	// OCTAL without notations
	result := stringBuilder.Reset()
		.AddAnyBit(
			anyBit := lwordVar, 
			option := E_AddAnyBitOptions.OCTAL, 
			lowerCase := FALSE, 
			displayedDigitsCount := 64, 
			addNotation := FALSE)
		.Create();
		
	AssertEquals_STRING(
		Actual := result,
		Expected := '0000000000000000000000000000000000000000000000000000000000000253',
		Message := 'Adding lword as OCTAL with addNotation = FALSE was incorrect');
		
	TcUnit.TEST_FINISHED();
END_IF
END_METHOD

METHOD Test28_ANY_REAL_REAL
VAR
	realVar	: REAL := 12345.123888;
	result	: Tc2_System.T_MaxString;
END_VAR
IF TcUnit.TEST_ORDERED('Test28_ANY_REAL_REAL') THEN
	result := stringBuilder.Reset().
		AddAnyReal(
			anyReal := realVar,
			precision := 2,
			round := FALSE)
		.Create();	

	AssertEquals_STRING(
		Actual := result,
		Expected := '12345.12',
		Message := 'Adding REAL with round = FALSE failed.');
		
	result := stringBuilder.Reset().
		AddAnyReal(
			anyReal := realVar,
			precision := 3,
			round := TRUE)
		.Create();	

	AssertEquals_STRING(
		Actual := result,
		Expected := '12345.124',
		Message := 'Adding REAL with round = TRUE failed.');
		
	TcUnit.TEST_FINISHED();
END_IF
END_METHOD

METHOD Test29_ANY_REAL_LREAL
VAR
	lrealVar	: LREAL := 12345.12345678;
	result	: Tc2_System.T_MaxString;
END_VAR
IF TcUnit.TEST_ORDERED('Test29_ANY_REAL_LREAL') THEN
	result := stringBuilder.Reset().
		AddAnyReal(
			anyReal := lrealVar,
			precision := 5,
			round := FALSE)
		.Create();	

	AssertEquals_STRING(
		Actual := result,
		Expected := '12345.12345',
		Message := 'Adding LREAL with round = FALSE failed.');
		
	result := stringBuilder.Reset().
		AddAnyReal(
			anyReal := lrealVar,
			precision := 7,
			round := TRUE)
		.Create();	

	AssertEquals_STRING(
		Actual := result,
		Expected := '12345.1234568',
		Message := 'Adding LREAL with round = TRUE failed.');
		
	TcUnit.TEST_FINISHED();
END_IF
END_METHOD

END_FUNCTION_BLOCK

// ---- TESTS/Test suites/FB_HasTaskInfo_Tests.TcPOU
FUNCTION_BLOCK internal FB_HasTaskInfo_Tests EXTENDS FB_TestSuite
VAR_INPUT
END_VAR
VAR_OUTPUT
END_VAR
VAR
END_VAR

Test01_TaskInfoPropertyValidity();

METHOD Test01_TaskInfoPropertyValidity
VAR_INPUT
END_VAR
VAR_INST
	fbTaskInfo	: FB_HasTaskInfo_ExtensionsForTests;
	cycles	: UINT;
END_VAR
TcUnit.TEST('Test01_TaskInfoPropertyValidity');

AssertTrue(
	Condition := __ISVALIDREF(fbTaskInfo.TaskInfo),
	Message := 'Invalid reference for Taskinfo property. PLC crash will occur if called!');
	
AssertTrue(
	Condition := fbTaskInfo.TaskInfo.AdsPort <> 0,
	Message := 'TaskInfo property is empty.');


TcUnit.TEST_FINISHED();
END_METHOD

END_FUNCTION_BLOCK

// ---- TESTS/Test suites/FB_HasTaskInfo_ExtensionsForTests.TcPOU
// Since FB_HasTaskInfo is an ABSTRACT class, the functionality needs to be implemented by extending the base class
FUNCTION_BLOCK internal FB_HasTaskInfo_ExtensionsForTests EXTENDS FB_HasTaskInfo
VAR_INPUT
END_VAR
VAR_OUTPUT
END_VAR
VAR
END_VAR

END_FUNCTION_BLOCK

// ---- SOURCE/General/FB_HasTaskInfo.TcPOU
{attribute 'no_explicit_call' := 'Body contains no logic, calling methods only allowed.'}
FUNCTION_BLOCK ABSTRACT FB_HasTaskInfo
VAR
	_PlcTaskInfo	: REFERENCE TO PlcTaskSystemInfo;
END_VAR

{attribute 'monitoring':='call'}
PROPERTY TaskInfo : REFERENCE TO PlcTaskSystemInfo
GET
VAR
	taskIndex	: DINT;
END_VAR
IF NOT __ISVALIDREF(_plcTaskInfo) OR_ELSE _plcTaskInfo.CycleTime = 0 THEN
	taskIndex := Tc2_System.GETCURTASKINDEXEX();
	IF taskIndex <> 0 THEN
		_PlcTaskInfo REF= TwinCAT_SystemInfoVarList._TaskInfo[taskIndex];
	END_IF
END_IF

TaskInfo REF= _PlcTaskInfo;
END_GET
END_PROPERTY

END_FUNCTION_BLOCK

// ---- TESTS/Test suites/FB_BoolEx_Tests.TcPOU
FUNCTION_BLOCK INTERNAL FB_BoolEx_Tests EXTENDS FB_TestSuite
VAR_INPUT
END_VAR
VAR_OUTPUT
END_VAR
VAR
	_boolVariable	: BOOL;
	_intVariable	: INT;
	_boolEx			: BoolEx := (variable := _boolVariable);
END_VAR

Test01_BooleanTrue_ExpectTrueAfterElapsedTime();
Test02_BooleanFalse_ExpectTrueAfterElapsedTime();
Test03_RisingAndFallingEdge_ExpectPulses();
Test04_GetAndSetValue();
Test05_Toggle_ExpectValueInverts();
Test06_PulseWithInterval_100ms_ExpectValueChangeEvery100ms();
Test07_Set_ExpectTrue();
Test08_Reset_ExpectFalse();

METHOD Test01_BooleanTrue_ExpectTrueAfterElapsedTime
VAR_INPUT
		
END_VAR
VAR_INST
	boolEx				: BoolEx := (variable := _boolVariable);
	conditionTrueTimer	: Tc2_Standard.TON;
END_VAR
TcUnit.TEST('Test01_BooleanTrue_ExpectTrueAfterElapsedTime');

conditionTrueTimer();
IF NOT conditionTrueTimer.Q THEN
	_boolVariable := TRUE;
	conditionTrueTimer(IN := TRUE, PT := T#20MS);
	AssertFalse(
		Condition := boolEx.HasBeenTrueForAtLeast(T#20MS),
		Message := 'HasBeenTrueForAtLeast returned TRUE before elapsed time.');
ELSE
	AssertTrue(
		Condition := boolEx.HasBeenTrueForAtLeast(T#20MS),
		Message := 'HasBeenTrueForAtLeast returned FALSE after elapsed time.');
		TcUnit.TEST_FINISHED();
END_IF
END_METHOD

METHOD Test02_BooleanFalse_ExpectTrueAfterElapsedTime : BOOL
VAR_INST
	boolEx			: BoolEx := (variable := _boolVariable);
	conditionTimer	: Tc2_Standard.TON;
END_VAR
TcUnit.TEST('Test02_BooleanFalse_ExpectTrueAfterElapsedTime');
IF TcUnit.IS_TEST_FINISHED('Test01_BooleanTrue_ExpectTrueAfterElapsedTime') THEN
	_boolVariable := FALSE;
	conditionTimer();
	IF NOT conditionTimer.Q THEN
		conditionTimer(IN := TRUE, PT := T#20MS);
		AssertFalse(
			Condition := boolEx.HasBeenFalseForAtLeast(T#20MS),
			Message := 'HasBeenFalseForAtLeast returned TRUE before elapsed time.');
	ELSE
		AssertTrue(
			Condition := boolEx.HasBeenFalseForAtLeast(T#20MS),
			Message := 'HasBeenFalseForAtLeast returned FALSE after elapsed time.');
			TcUnit.TEST_FINISHED();
	END_IF
END_IF
END_METHOD

METHOD Test03_RisingAndFallingEdge_ExpectPulses
VAR_INPUT
END_VAR

VAR_INST
	boolEx : BoolEx := (variable := _boolVariable);
END_VAR
TcUnit.TEST('Test03_RisingAndFallingEdge_ExpectPulses');


IF TcUnit.IS_TEST_FINISHED('Test02_BooleanFalse_ExpectTrueAfterElapsedTime') THEN
	_boolVariable := FALSE;
	AssertFalse(
		Condition := boolEx.HasRisingEdge,
		Message := 'When value has not changed, the HasRisingEdge should be false');
	AssertFalse(
		Condition := boolEx.HasFallingEdge,
		Message := 'When value has not changed, the HasFallingEdge should be false');
	_boolVariable := TRUE;	
	AssertTrue(
		Condition := boolEx.HasRisingEdge,
		Message := 'When value has changed from FALSE to TRUE, the HasRisingEdge should be TRUE');
	AssertFalse(
		Condition := boolEx.HasFallingEdge,
		Message := 'When value has changed to TRUE, the HasFallingEdge should be false');
	_boolVariable := FALSE;
	AssertTrue(
		Condition := boolEx.HasFallingEdge,
		Message := 'When value has changed from TRUE to FALSE, the HasFallingEdge should be TRUE');
	AssertFalse(
		Condition := boolEx.HasRisingEdge,
		Message := 'When value has not changed, the HasRisingEdge should be false');
	AssertFalse(
		Condition := boolEx.HasFallingEdge,
		Message := 'When value has not changed, the HasRisingEdge should be false');	
	TcUnit.TEST_FINISHED();
	
END_IF
END_METHOD

METHOD Test04_GetAndSetValue
VAR_INPUT
END_VAR
VAR_INST
	boolEx	: BoolEx := (variable := _boolVariable);
END_VAR
TcUnit.TEST('Test04_GetAndSetValue');
IF TcUnit.IS_TEST_FINISHED('Test03_RisingAndFallingEdge_ExpectPulses') THEN
	_boolVariable := FALSE;
	boolEx.Value := TRUE;	
	AssertTrue(
		Condition := _boolVariable,
		Message := 'Setting value to TRUE failed');
		
	boolEx.Value := FALSE;
	AssertFalse(
		Condition := _boolVariable,
		Message := 'Setting value to FALSE failed');
		
	AssertEquals_BOOL(
		Actual := boolEx.Value,
		Expected := _boolVariable,
		Message := 'Value returned incorrect result.');
		
	_boolVariable := TRUE;
	AssertEquals_BOOL(
		Actual := boolEx.Value,
		Expected := _boolVariable,
		Message := 'Value returned incorrect result.');
	
	TcUnit.TEST_FINISHED();
END_IF
END_METHOD

METHOD Test05_Toggle_ExpectValueInverts
VAR_INPUT
END_VAR
TcUnit.TEST('Test05_Toggle_ExpectValueInverts');
IF TcUnit.IS_TEST_FINISHED('Test04_GetAndSetValue') THEN
	_boolEx.Value := FALSE;
	AssertFalse(
		Condition := _boolEx.Value,
		Message := 'Expected value to be false.');
		
	_boolEx.Toggle();
	AssertTrue(
		Condition := _boolEx.Value,
		Message := 'Toggle to TRUE failed');
		
	_boolEx.Toggle();
	AssertFalse(
		Condition := _boolEx.Value,
		Message := 'Toggle to FALSE failed');	
	TcUnit.TEST_FINISHED();
END_IF
END_METHOD

METHOD Test06_PulseWithInterval_100ms_ExpectValueChangeEvery100ms
VAR_INPUT
END_VAR
VAR_INST
	timerOn		: Tc2_Standard.TON;
	timerOff	: Tc2_Standard.TON;
END_VAR
TcUnit.TEST('Test06_PulseWithInterval_100ms_ExpectValueChangeEvery100ms');
IF TcUnit.IS_TEST_FINISHED('Test05_Toggle_ExpectValueInverts') THEN
	_boolEx.Value := FALSE;
	_boolEx.PulseWithInterval(durationOn := T#100MS, durationOff := T#50MS);
	timerOn(IN := TRUE, PT := T#100MS);
	IF NOT timerOn.Q THEN
		AssertTrue(
			Condition := _boolEx.Value,
			Message := 'Value should be TRUE until the durationOn expires.');
	ELSE
		timerOff(IN := TRUE, PT := T#50MS);
		IF timeroff.Q THEN
			AssertTrue(
				Condition := _boolEx.Value,
				Message := 'Value should be TRUE after the durationOff expires.');
			TcUnit.TEST_FINISHED();
			RETURN;
		END_IF
		AssertFalse(
			Condition := _boolEx.Value,
			Message := 'Value should be FALSE after durationOn expires.');

	END_IF
END_IF
END_METHOD

METHOD Test07_Set_ExpectTrue
VAR_INPUT
END_VAR
TcUnit.TEST('Test07_Set_ExpectTrue');

IF TcUnit.IS_TEST_FINISHED('Test06_PulseWithInterval_100ms_ExpectValueChangeEvery100ms') THEN 
	_boolEx.Value := FALSE;
	_boolEx.Set();
	AssertTrue(
		Condition := _boolEx.Value,
		Message := 'Set() did not set the value to TRUE.');
	TcUnit.TEST_FINISHED();
END_IF
END_METHOD

METHOD Test08_Reset_ExpectFalse
VAR_INPUT
END_VAR
TcUnit.TEST('Test08_Reset_ExpectFalse');

IF TcUnit.IS_TEST_FINISHED('Test07_Set_ExpectTrue') THEN 
	_boolEx.Value := TRUE;
	_boolEx.Reset();
	AssertFalse(
		Condition := _boolEx.Value,
		Message := 'Reset() did not set the value to FALSE.');
	TcUnit.TEST_FINISHED();
END_IF
END_METHOD

END_FUNCTION_BLOCK

// ---- SOURCE/General/Variable extensions/BoolEx.TcPOU
// An extension to boolean variable
FUNCTION_BLOCK BoolEx
VAR_INPUT
	variable			: REFERENCE TO BOOL;
END_VAR

VAR
	
	_risingEdge			: Tc2_Standard.R_TRIG;
	_fallingEdge		: Tc2_Standard.F_TRIG;
	afterinitvarinfo 	: ST_VarInfo;
END_VAR

// Returns TRUE if monitored value has been FALSE for at lease for the provided "duration"
METHOD HasBeenFalseForAtLeast : BOOL
VAR_INPUT
	duration	: TIME;
END_VAR

VAR_INST
	timer	: Tc2_Standard.TON;

END_VAR
IF NOT IsVarValid() THEN
	RETURN;
END_IF

timer(IN := NOT variable, PT := duration);
HasBeenFalseForAtLeast := timer.Q;
END_METHOD

// Returns TRUE if monitored value has been TRUE for at lease for the provided "duration"
METHOD HasBeenTrueForAtLeast : BOOL
VAR_INPUT
	duration	: TIME;
END_VAR

VAR_INST
	timer	: Tc2_Standard.TON;
	ptrBool	: POINTER TO BOOL;
END_VAR
IF NOT IsVarValid() THEN
	RETURN;
END_IF

timer(IN := variable, PT := duration);
HasBeenTrueForAtLeast := timer.Q;
END_METHOD

// Returns TRUE if oberved variable change from TRUE to FALSE from the last call.
PROPERTY HasFallingEdge : BOOL
GET
_fallingEdge(CLK := variable);
HasFallingEdge := _fallingEdge.Q;
END_GET
END_PROPERTY

// Returns TRUE if oberved variable change from FALSE to TRUE from the last call.
PROPERTY HasRisingEdge : BOOL
GET
_risingEdge(CLK := variable);
HasRisingEdge := _risingEdge.Q;
END_GET
END_PROPERTY

METHOD PROTECTED IsVarValid : BOOL
IsVarValid := __ISVALIDREF(variable);
END_METHOD

// Pulses the virabile (TRUE/FALSE) with the provided on and off duration
METHOD PulseWithInterval
VAR_INPUT
	durationOn	: TIME;
	durationOff	: TIME;
END_VAR
VAR_INST
	timerOn		: Tc2_Standard.TON;
	timerOff	: Tc2_Standard.TON;
END_VAR
IF NOT IsVarValid() THEN
	RETURN;
END_IF
// In order to properly trigger immediate change, call both timers twice. 
// This way when ON is elapsed, OFF starts imediately and vice versa.
timerOff(IN := timerOn.Q, PT := durationOff);
timerOn(IN := NOT timerOff.Q, PT := durationOn);
timerOff(IN := timerOn.Q, PT := durationOff);
timerOn(IN := NOT timerOff.Q, PT := durationOn);
variable := NOT timerOn.Q;
END_METHOD

// Sets the value to FALSE
METHOD Reset
VAR_INPUT
END_VAR
IF NOT IsVarValid() THEN
	RETURN;
END_IF

variable := FALSE;
END_METHOD

// Sets the value to TRUE
METHOD Set
VAR_INPUT
END_VAR
IF NOT IsVarValid() THEN
	RETURN;
END_IF

variable := TRUE;
END_METHOD

METHOD Toggle
IF NOT IsVarValid() THEN
	RETURN;
END_IF

variable := NOT variable;
END_METHOD

PROPERTY Value : BOOL
GET
Value := variable;
END_GET
SET
variable := Value;
END_SET
END_PROPERTY

END_FUNCTION_BLOCK

// ---- TESTS/Test suites/FB_EthercatHelper_Tests.TcPOU
FUNCTION_BLOCK INTERNAL FB_EthercatHelper_Tests EXTENDS FB_TestSuite
VAR_INPUT
END_VAR
VAR_OUTPUT
END_VAR
VAR
END_VAR

Test01_ConvertBeckhoffEcState_ProvideAllOptions_ExpectCorrectResults();

METHOD Test01_ConvertBeckhoffEcState_ProvideAllOptions_ExpectCorrectResults
VAR_INST
	ecSlaveState		: Tc2_EtherCAT.ST_EcSlaveState;
	helperEcSlaveState	: ST_EcSlaveState;
END_VAR
TcUnit.TEST('Test01_ConvertBeckhoffEcState_ProvideAllOptions_ExpectCorrectResults');

// Init
ecSlaveState.deviceState := Tc2_EtherCAT.EC_DEVICE_STATE_INIT;
helperEcSlaveState := EthercatHelper.ConvertBeckhoffEcStateToCustomStruct(ecSlaveState);
AssertEquals_BYTE(Tc2_EtherCAT.EC_DEVICE_STATE_INIT, helperEcSlaveState.Device.State, 'Incorrect state for EC_DEVICE_STATE_INIT.');
AssertEquals_BYTE(E_EcDeviceStateExtras.NOTHING, helperEcSlaveState.Device.StateExtras, 'EC_DEVICE_STATE_INIT - Extras NOTHING expected');
	
ecSlaveState.deviceState := Tc2_EtherCAT.EC_DEVICE_STATE_INIT OR Tc2_EtherCAT.EC_DEVICE_STATE_INITCMD_ERROR;
helperEcSlaveState := EthercatHelper.ConvertBeckhoffEcStateToCustomStruct(ecSlaveState);
AssertEquals_BYTE(Tc2_EtherCAT.EC_DEVICE_STATE_INIT, helperEcSlaveState.Device.State,'Incorrect state for EC_DEVICE_STATE_INIT OR EC_DEVICE_STATE_INITCMD_ERROR');
AssertEquals_BYTE(E_EcDeviceStateExtras.INIIT_CMD_ERROR, helperEcSlaveState.Device.StateExtras, 'EC_DEVICE_STATE_INIT - Extras INIIT_CMD_ERROR expected');
	
ecSlaveState.deviceState := Tc2_EtherCAT.EC_DEVICE_STATE_INIT OR Tc2_EtherCAT.EC_DEVICE_STATE_INVALID_VPRS;
helperEcSlaveState := EthercatHelper.ConvertBeckhoffEcStateToCustomStruct(ecSlaveState);
AssertEquals_BYTE(Tc2_EtherCAT.EC_DEVICE_STATE_INIT, helperEcSlaveState.Device.State,'Incorrect state for EC_DEVICE_STATE_INIT OR EC_DEVICE_STATE_INVALID_VPRS');
AssertEquals_BYTE(E_EcDeviceStateExtras.INVALID_VPRS, helperEcSlaveState.Device.StateExtras, 'EC_DEVICE_STATE_INIT - Extras INVALID_VPRS expected');

ecSlaveState.deviceState := Tc2_EtherCAT.EC_DEVICE_STATE_INIT OR Tc2_EtherCAT.EC_DEVICE_STATE_DISABLED;
helperEcSlaveState := EthercatHelper.ConvertBeckhoffEcStateToCustomStruct(ecSlaveState);
AssertEquals_BYTE(Tc2_EtherCAT.EC_DEVICE_STATE_INIT, helperEcSlaveState.Device.State,'Incorrect state for EC_DEVICE_STATE_INIT OR EC_DEVICE_STATE_DISABLED');
AssertEquals_BYTE(E_EcDeviceStateExtras.DISABLED, helperEcSlaveState.Device.StateExtras, 'EC_DEVICE_STATE_INIT - Extras DISABLED expected');

ecSlaveState.deviceState := Tc2_EtherCAT.EC_DEVICE_STATE_INIT OR Tc2_EtherCAT.EC_DEVICE_STATE_ERROR;
helperEcSlaveState := EthercatHelper.ConvertBeckhoffEcStateToCustomStruct(ecSlaveState);
AssertEquals_BYTE(Tc2_EtherCAT.EC_DEVICE_STATE_INIT, helperEcSlaveState.Device.State,'Incorrect state for EC_DEVICE_STATE_INIT OR EC_DEVICE_STATE_ERROR');
AssertEquals_BYTE(E_EcDeviceStateExtras.STATE_MACHINE_ERROR, helperEcSlaveState.Device.StateExtras, 'EC_DEVICE_STATE_INIT - Extras STATE_MACHINE_ERROR expected');
	
// Pre-op
ecSlaveState.deviceState := Tc2_EtherCAT.EC_DEVICE_STATE_PREOP;
helperEcSlaveState := EthercatHelper.ConvertBeckhoffEcStateToCustomStruct(ecSlaveState);
AssertEquals_BYTE(Tc2_EtherCAT.EC_DEVICE_STATE_PREOP, helperEcSlaveState.Device.State, 'Incorrect state for EC_DEVICE_STATE_PREOP.');
AssertEquals_BYTE(E_EcDeviceStateExtras.NOTHING, helperEcSlaveState.Device.StateExtras, 'EC_DEVICE_STATE_PREOP - Extras NOTHING expected');
	
ecSlaveState.deviceState := Tc2_EtherCAT.EC_DEVICE_STATE_PREOP OR Tc2_EtherCAT.EC_DEVICE_STATE_INITCMD_ERROR;
helperEcSlaveState := EthercatHelper.ConvertBeckhoffEcStateToCustomStruct(ecSlaveState);
AssertEquals_BYTE(Tc2_EtherCAT.EC_DEVICE_STATE_PREOP, helperEcSlaveState.Device.State,'Incorrect state for EC_DEVICE_STATE_PREOP OR EC_DEVICE_STATE_INITCMD_ERROR');
AssertEquals_BYTE(E_EcDeviceStateExtras.INIIT_CMD_ERROR, helperEcSlaveState.Device.StateExtras, 'EC_DEVICE_STATE_PREOP - Extras INIIT_CMD_ERROR expected');
	
ecSlaveState.deviceState := Tc2_EtherCAT.EC_DEVICE_STATE_PREOP OR Tc2_EtherCAT.EC_DEVICE_STATE_INVALID_VPRS;
helperEcSlaveState := EthercatHelper.ConvertBeckhoffEcStateToCustomStruct(ecSlaveState);
AssertEquals_BYTE(Tc2_EtherCAT.EC_DEVICE_STATE_PREOP, helperEcSlaveState.Device.State,'Incorrect state for EC_DEVICE_STATE_PREOP OR EC_DEVICE_STATE_INVALID_VPRS');
AssertEquals_BYTE(E_EcDeviceStateExtras.INVALID_VPRS, helperEcSlaveState.Device.StateExtras, 'EC_DEVICE_STATE_PREOP - Extras INVALID_VPRS expected');

ecSlaveState.deviceState := Tc2_EtherCAT.EC_DEVICE_STATE_PREOP OR Tc2_EtherCAT.EC_DEVICE_STATE_DISABLED;
helperEcSlaveState := EthercatHelper.ConvertBeckhoffEcStateToCustomStruct(ecSlaveState);
AssertEquals_BYTE(Tc2_EtherCAT.EC_DEVICE_STATE_PREOP, helperEcSlaveState.Device.State,'Incorrect state for EC_DEVICE_STATE_PREOP OR EC_DEVICE_STATE_DISABLED');
AssertEquals_BYTE(E_EcDeviceStateExtras.DISABLED, helperEcSlaveState.Device.StateExtras, 'EC_DEVICE_STATE_PREOP - Extras DISABLED expected');

ecSlaveState.deviceState := Tc2_EtherCAT.EC_DEVICE_STATE_PREOP OR Tc2_EtherCAT.EC_DEVICE_STATE_ERROR;
helperEcSlaveState := EthercatHelper.ConvertBeckhoffEcStateToCustomStruct(ecSlaveState);
AssertEquals_BYTE(Tc2_EtherCAT.EC_DEVICE_STATE_PREOP, helperEcSlaveState.Device.State,'Incorrect state for EC_DEVICE_STATE_PREOP OR EC_DEVICE_STATE_ERROR');
AssertEquals_BYTE(E_EcDeviceStateExtras.STATE_MACHINE_ERROR, helperEcSlaveState.Device.StateExtras, 'EC_DEVICE_STATE_PREOP - Extras STATE_MACHINE_ERROR expected');

// Bootstrap
ecSlaveState.deviceState := Tc2_EtherCAT.EC_DEVICE_STATE_BOOTSTRAP;
helperEcSlaveState := EthercatHelper.ConvertBeckhoffEcStateToCustomStruct(ecSlaveState);
AssertEquals_BYTE(Tc2_EtherCAT.EC_DEVICE_STATE_BOOTSTRAP, helperEcSlaveState.Device.State, 'Incorrect state for EC_DEVICE_STATE_BOOTSTRAP.');
AssertEquals_BYTE(E_EcDeviceStateExtras.NOTHING, helperEcSlaveState.Device.StateExtras, 'EC_DEVICE_STATE_BOOTSTRAP - Extras NOTHING expected');
	
ecSlaveState.deviceState := Tc2_EtherCAT.EC_DEVICE_STATE_BOOTSTRAP OR Tc2_EtherCAT.EC_DEVICE_STATE_INITCMD_ERROR;
helperEcSlaveState := EthercatHelper.ConvertBeckhoffEcStateToCustomStruct(ecSlaveState);
AssertEquals_BYTE(Tc2_EtherCAT.EC_DEVICE_STATE_BOOTSTRAP, helperEcSlaveState.Device.State,'Incorrect state for EC_DEVICE_STATE_BOOTSTRAP OR EC_DEVICE_STATE_INITCMD_ERROR');
AssertEquals_BYTE(E_EcDeviceStateExtras.INIIT_CMD_ERROR, helperEcSlaveState.Device.StateExtras, 'EC_DEVICE_STATE_BOOTSTRAP - Extras INIIT_CMD_ERROR expected');
	
ecSlaveState.deviceState := Tc2_EtherCAT.EC_DEVICE_STATE_BOOTSTRAP OR Tc2_EtherCAT.EC_DEVICE_STATE_INVALID_VPRS;
helperEcSlaveState := EthercatHelper.ConvertBeckhoffEcStateToCustomStruct(ecSlaveState);
AssertEquals_BYTE(Tc2_EtherCAT.EC_DEVICE_STATE_BOOTSTRAP, helperEcSlaveState.Device.State,'Incorrect state for EC_DEVICE_STATE_BOOTSTRAP OR EC_DEVICE_STATE_INVALID_VPRS');
AssertEquals_BYTE(E_EcDeviceStateExtras.INVALID_VPRS, helperEcSlaveState.Device.StateExtras, 'EC_DEVICE_STATE_BOOTSTRAP - Extras INVALID_VPRS expected');

ecSlaveState.deviceState := Tc2_EtherCAT.EC_DEVICE_STATE_BOOTSTRAP OR Tc2_EtherCAT.EC_DEVICE_STATE_DISABLED;
helperEcSlaveState := EthercatHelper.ConvertBeckhoffEcStateToCustomStruct(ecSlaveState);
AssertEquals_BYTE(Tc2_EtherCAT.EC_DEVICE_STATE_BOOTSTRAP, helperEcSlaveState.Device.State,'Incorrect state for EC_DEVICE_STATE_BOOTSTRAP OR EC_DEVICE_STATE_DISABLED');
AssertEquals_BYTE(E_EcDeviceStateExtras.DISABLED, helperEcSlaveState.Device.StateExtras, 'EC_DEVICE_STATE_BOOTSTRAP - Extras DISABLED expected');

ecSlaveState.deviceState := Tc2_EtherCAT.EC_DEVICE_STATE_BOOTSTRAP OR Tc2_EtherCAT.EC_DEVICE_STATE_ERROR;
helperEcSlaveState := EthercatHelper.ConvertBeckhoffEcStateToCustomStruct(ecSlaveState);
AssertEquals_BYTE(Tc2_EtherCAT.EC_DEVICE_STATE_BOOTSTRAP, helperEcSlaveState.Device.State,'Incorrect state for EC_DEVICE_STATE_BOOTSTRAP OR EC_DEVICE_STATE_ERROR');
AssertEquals_BYTE(E_EcDeviceStateExtras.STATE_MACHINE_ERROR, helperEcSlaveState.Device.StateExtras, 'EC_DEVICE_STATE_BOOTSTRAP - Extras STATE_MACHINE_ERROR expected');

// Safeop
ecSlaveState.deviceState := Tc2_EtherCAT.EC_DEVICE_STATE_SAFEOP;
helperEcSlaveState := EthercatHelper.ConvertBeckhoffEcStateToCustomStruct(ecSlaveState);
AssertEquals_BYTE(Tc2_EtherCAT.EC_DEVICE_STATE_SAFEOP, helperEcSlaveState.Device.State, 'Incorrect state for EC_DEVICE_STATE_SAFEOP.');
AssertEquals_BYTE(E_EcDeviceStateExtras.NOTHING, helperEcSlaveState.Device.StateExtras, 'EC_DEVICE_STATE_SAFEOP - Extras NOTHING expected');
	
ecSlaveState.deviceState := Tc2_EtherCAT.EC_DEVICE_STATE_SAFEOP OR Tc2_EtherCAT.EC_DEVICE_STATE_INITCMD_ERROR;
helperEcSlaveState := EthercatHelper.ConvertBeckhoffEcStateToCustomStruct(ecSlaveState);
AssertEquals_BYTE(Tc2_EtherCAT.EC_DEVICE_STATE_SAFEOP, helperEcSlaveState.Device.State,'Incorrect state for EC_DEVICE_STATE_BOOTSTRAP OR EC_DEVICE_STATE_INITCMD_ERROR');
AssertEquals_BYTE(E_EcDeviceStateExtras.INIIT_CMD_ERROR, helperEcSlaveState.Device.StateExtras, 'EC_DEVICE_STATE_SAFEOP - Extras INIIT_CMD_ERROR expected');
	
ecSlaveState.deviceState := Tc2_EtherCAT.EC_DEVICE_STATE_SAFEOP OR Tc2_EtherCAT.EC_DEVICE_STATE_INVALID_VPRS;
helperEcSlaveState := EthercatHelper.ConvertBeckhoffEcStateToCustomStruct(ecSlaveState);
AssertEquals_BYTE(Tc2_EtherCAT.EC_DEVICE_STATE_SAFEOP, helperEcSlaveState.Device.State,'Incorrect state for EC_DEVICE_STATE_SAFEOP OR EC_DEVICE_STATE_INVALID_VPRS');
AssertEquals_BYTE(E_EcDeviceStateExtras.INVALID_VPRS, helperEcSlaveState.Device.StateExtras, 'EC_DEVICE_STATE_SAFEOP - Extras INVALID_VPRS expected');

ecSlaveState.deviceState := Tc2_EtherCAT.EC_DEVICE_STATE_SAFEOP OR Tc2_EtherCAT.EC_DEVICE_STATE_DISABLED;
helperEcSlaveState := EthercatHelper.ConvertBeckhoffEcStateToCustomStruct(ecSlaveState);
AssertEquals_BYTE(Tc2_EtherCAT.EC_DEVICE_STATE_SAFEOP, helperEcSlaveState.Device.State,'Incorrect state for EC_DEVICE_STATE_SAFEOP OR EC_DEVICE_STATE_DISABLED');
AssertEquals_BYTE(E_EcDeviceStateExtras.DISABLED, helperEcSlaveState.Device.StateExtras, 'EC_DEVICE_STATE_SAFEOP - Extras DISABLED expected');

ecSlaveState.deviceState := Tc2_EtherCAT.EC_DEVICE_STATE_SAFEOP OR Tc2_EtherCAT.EC_DEVICE_STATE_ERROR;
helperEcSlaveState := EthercatHelper.ConvertBeckhoffEcStateToCustomStruct(ecSlaveState);
AssertEquals_BYTE(Tc2_EtherCAT.EC_DEVICE_STATE_SAFEOP, helperEcSlaveState.Device.State,'Incorrect state for EC_DEVICE_STATE_SAFEOP OR EC_DEVICE_STATE_ERROR');
AssertEquals_BYTE(E_EcDeviceStateExtras.STATE_MACHINE_ERROR, helperEcSlaveState.Device.StateExtras, 'EC_DEVICE_STATE_SAFEOP - Extras STATE_MACHINE_ERROR expected');

// OP
ecSlaveState.deviceState := Tc2_EtherCAT.EC_DEVICE_STATE_OP;
helperEcSlaveState := EthercatHelper.ConvertBeckhoffEcStateToCustomStruct(ecSlaveState);
AssertEquals_BYTE(Tc2_EtherCAT.EC_DEVICE_STATE_OP, helperEcSlaveState.Device.State, 'Incorrect state for EC_DEVICE_STATE_OP.');
AssertEquals_BYTE(E_EcDeviceStateExtras.NOTHING, helperEcSlaveState.Device.StateExtras, 'EC_DEVICE_STATE_OP - Extras NOTHING expected');
	
ecSlaveState.deviceState := Tc2_EtherCAT.EC_DEVICE_STATE_OP OR Tc2_EtherCAT.EC_DEVICE_STATE_INITCMD_ERROR;
helperEcSlaveState := EthercatHelper.ConvertBeckhoffEcStateToCustomStruct(ecSlaveState);
AssertEquals_BYTE(Tc2_EtherCAT.EC_DEVICE_STATE_OP, helperEcSlaveState.Device.State,'Incorrect state for EC_DEVICE_STATE_OP OR EC_DEVICE_STATE_INITCMD_ERROR');
AssertEquals_BYTE(E_EcDeviceStateExtras.INIIT_CMD_ERROR, helperEcSlaveState.Device.StateExtras, 'EC_DEVICE_STATE_OP - Extras INIIT_CMD_ERROR expected');
	
ecSlaveState.deviceState := Tc2_EtherCAT.EC_DEVICE_STATE_OP OR Tc2_EtherCAT.EC_DEVICE_STATE_INVALID_VPRS;
helperEcSlaveState := EthercatHelper.ConvertBeckhoffEcStateToCustomStruct(ecSlaveState);
AssertEquals_BYTE(Tc2_EtherCAT.EC_DEVICE_STATE_OP, helperEcSlaveState.Device.State,'Incorrect state for EC_DEVICE_STATE_OP OR EC_DEVICE_STATE_INVALID_VPRS');
AssertEquals_BYTE(E_EcDeviceStateExtras.INVALID_VPRS, helperEcSlaveState.Device.StateExtras, 'EC_DEVICE_STATE_OP - Extras INVALID_VPRS expected');

ecSlaveState.deviceState := Tc2_EtherCAT.EC_DEVICE_STATE_OP OR Tc2_EtherCAT.EC_DEVICE_STATE_DISABLED;
helperEcSlaveState := EthercatHelper.ConvertBeckhoffEcStateToCustomStruct(ecSlaveState);
AssertEquals_BYTE(Tc2_EtherCAT.EC_DEVICE_STATE_OP, helperEcSlaveState.Device.State,'Incorrect state for EC_DEVICE_STATE_OP OR EC_DEVICE_STATE_DISABLED');
AssertEquals_BYTE(E_EcDeviceStateExtras.DISABLED, helperEcSlaveState.Device.StateExtras, 'EC_DEVICE_STATE_OP - Extras DISABLED expected');

ecSlaveState.deviceState := Tc2_EtherCAT.EC_DEVICE_STATE_OP OR Tc2_EtherCAT.EC_DEVICE_STATE_ERROR;
helperEcSlaveState := EthercatHelper.ConvertBeckhoffEcStateToCustomStruct(ecSlaveState);
AssertEquals_BYTE(Tc2_EtherCAT.EC_DEVICE_STATE_OP, helperEcSlaveState.Device.State,'Incorrect state for EC_DEVICE_STATE_OP OR EC_DEVICE_STATE_ERROR');
AssertEquals_BYTE(E_EcDeviceStateExtras.STATE_MACHINE_ERROR, helperEcSlaveState.Device.StateExtras, 'EC_DEVICE_STATE_OP - Extras STATE_MACHINE_ERROR expected');

// Link state

//EC_LINK_STATE_OK
ecSlaveState.linkState := Tc2_EtherCAT.EC_LINK_STATE_OK;
helperEcSlaveState := EthercatHelper.ConvertBeckhoffEcStateToCustomStruct(ecSlaveState);
AssertEquals_BYTE(Tc2_EtherCAT.EC_LINK_STATE_OK, helperEcSlaveState.Link, 'Invalid link state for EC_LINK_STATE_OK');

// EC_LINK_STATE_ADDITIONAL_LINK
ecSlaveState.linkState := Tc2_EtherCAT.EC_LINK_STATE_ADDITIONAL_LINK;
helperEcSlaveState := EthercatHelper.ConvertBeckhoffEcStateToCustomStruct(ecSlaveState);
AssertEquals_BYTE(E_EcLinkState.ADDITIONAL_LINK, helperEcSlaveState.Link, 'Invalid link state for EC_LINK_STATE_ADDITIONAL_LINK');

// EC_LINK_STATE_LINK_WITHOUT_COMM
ecSlaveState.linkState := Tc2_EtherCAT.EC_LINK_STATE_LINK_WITHOUT_COMM;
helperEcSlaveState := EthercatHelper.ConvertBeckhoffEcStateToCustomStruct(ecSlaveState);
AssertEquals_BYTE(E_EcLinkState.LINK_WITHOUT_COMM, helperEcSlaveState.Link, 'Invalid link state for EC_LINK_STATE_LINK_WITHOUT_COMM');

// EC_LINK_STATE_MISSING_LINK
ecSlaveState.linkState := Tc2_EtherCAT.EC_LINK_STATE_MISSING_LINK;
helperEcSlaveState := EthercatHelper.ConvertBeckhoffEcStateToCustomStruct(ecSlaveState);
AssertEquals_BYTE(E_EcLinkState.MISSING_LINK, helperEcSlaveState.Link, 'Invalid link state for EC_LINK_STATE_MISSING_LINK');

// EC_LINK_STATE_NOT_PRESENT
ecSlaveState.linkState := Tc2_EtherCAT.EC_LINK_STATE_NOT_PRESENT;
helperEcSlaveState := EthercatHelper.ConvertBeckhoffEcStateToCustomStruct(ecSlaveState);
AssertEquals_BYTE(E_EcLinkState.NOT_PRESENT, helperEcSlaveState.Link, 'Invalid link state for EC_LINK_STATE_NOT_PRESENT');

// EC_LINK_STATE_PORT_A
ecSlaveState.linkState := Tc2_EtherCAT.EC_LINK_STATE_PORT_A;
helperEcSlaveState := EthercatHelper.ConvertBeckhoffEcStateToCustomStruct(ecSlaveState);
AssertEquals_BYTE(E_EcLinkState.PORT_A, helperEcSlaveState.Link, 'Invalid link state for EC_LINK_STATE_PORT_A');

// EC_LINK_STATE_PORT_B
ecSlaveState.linkState := Tc2_EtherCAT.EC_LINK_STATE_PORT_B;
helperEcSlaveState := EthercatHelper.ConvertBeckhoffEcStateToCustomStruct(ecSlaveState);
AssertEquals_BYTE(E_EcLinkState.PORT_B, helperEcSlaveState.Link, 'Invalid link state for EC_LINK_STATE_PORT_B');

// EC_LINK_STATE_PORT_C
ecSlaveState.linkState := Tc2_EtherCAT.EC_LINK_STATE_PORT_C;
helperEcSlaveState := EthercatHelper.ConvertBeckhoffEcStateToCustomStruct(ecSlaveState);
AssertEquals_BYTE(E_EcLinkState.PORT_C, helperEcSlaveState.Link, 'Invalid link state for EC_LINK_STATE_PORT_C');

// EC_LINK_STATE_PORT_D
ecSlaveState.linkState := Tc2_EtherCAT.EC_LINK_STATE_PORT_D;
helperEcSlaveState := EthercatHelper.ConvertBeckhoffEcStateToCustomStruct(ecSlaveState);
AssertEquals_BYTE(E_EcLinkState.PORT_D, helperEcSlaveState.Link, 'Invalid link state for EC_LINK_STATE_PORT_D');

TcUnit.TEST_FINISHED();
END_METHOD

END_FUNCTION_BLOCK

// ---- SOURCE/Beckhoff/EtherCAT/EthercatHelper.TcPOU
{attribute 'hide_all_locals'}
PROGRAM EthercatHelper
VAR
	fbReadDeviceName	: Tc2_IoFunctions.IOF_GetBoxNameByAddr;
	nMasterId			: UDINT;
END_VAR

// Converts Tc2_EtherCAT.ST_EcSlaveState to ZigaLibs_Core.ST_EcSlaveState and returns the converted structure.
METHOD ConvertBeckhoffEcStateToCustomStruct : ST_EcSlaveState
VAR_INPUT
	ecSlaveState	: Tc2_EtherCAT.ST_EcSlaveState;
END_VAR
VAR CONSTANT
	SLAVE_STATE_MASK 		: BYTE := 16#0F;
	SLAVE_STATE_EXTRAS_MASK : BYTE := 16#F0;
END_VAR
ConvertBeckhoffEcStateToCustomStruct.Device.State := SLAVE_STATE_MASK AND ecSlaveState.deviceState;
ConvertBeckhoffEcStateToCustomStruct.Device.StateExtras := SLAVE_STATE_EXTRAS_MASK AND ecSlaveState.deviceState;
ConvertBeckhoffEcStateToCustomStruct.Link := ecSlaveState.linkState;
END_METHOD

METHOD PUBLIC GetBoxNameByAddress : T_MaxString
VAR_INPUT
	PlcRuntimeNetId		: Tc2_System.T_AmsNetID; // NetId of the PLC where the devuce is located
	AmsNetId			: AMSADDR; // NetId of the box
	outError			: REFERENCE TO BOOL;	// If an error occurs while executing, method will provide the error flag here. This is a pointer to YOUR boolean error variable.
END_VAR

VAR
	sNetId	: Tc2_System.T_AmsNetID;
END_VAR
sNetId := AdsHelper.NetIdToString(AmsNetId.netId);
fbReadDeviceName(
	NETID := PlcRuntimeNetId,
	DEVICEID := AdsHelper.GetEthercatMasterIdFromNetIdString(netId := sNetId),
	BOXADDR := AmsNetId.port,
	START := NOT fbReadDeviceName.BUSY);
	
outError := fbReadDeviceName.ERR;
GetBoxNameByAddress := fbReadDeviceName.BOXNAME;
END_METHOD

END_PROGRAM

// ---- TESTS/Test suites/FB_Malloc_Tests.TcPOU
FUNCTION_BLOCK internal FB_Malloc_Tests EXTENDS FB_TestSuite
VAR_INPUT
END_VAR
VAR_OUTPUT
END_VAR
VAR
	_malloc							: FB_Malloc(0,0);
	_routerInfoBeforeTestMethod		: Tc2_Utilities.ST_TcRouterStatusInfo;
END_VAR

Test01_ProvideIncorrectParameters_ExpectNoAllocation();
Test02_Allocate10Integers_ExpectNoError_ValidateProperties();
Test03_Free_ExpectNoMemoryAllocated();
Test04_SetAndGet_ExpectGetReturnsCorrectValue();
Test05_SetAtIncorrectIndex_ExpectFalseReturned();
Test06_GetFromIncorrectIndex_ExpectTargetValueUnchanged_MethodReturnFalse();
Test07_Expand_ExpectOldDataStillExists_LastDataSetIsEmpty();
Test08_Remove_ExpectDataSetToCollapseBy1();

METHOD BeforeTestFinish : BOOL
VAR_INST
	currentRouterStatus	: Tc2_Utilities.ST_TcRouterStatusInfo;
END_VAR
_malloc.Free();
IF MemoryHelper.GetRouterStatusInfo('', currentRouterStatus) THEN
	AssertEquals_DWORD(
		Expected := _routerInfoBeforeTestMethod.maxMemAvail,
		Actual := currentRouterStatus.maxMemAvail,
		Message := 'The current and starting memory in router differ - memory leak detected.');
	BeforeTestFinish := TRUE;
END_IF
END_METHOD

METHOD BeforeTestStart : BOOL
VAR_INPUT
	methodName	: Tc2_System.T_MaxString;
END_VAR
VAR_INST
	previousMethodName	: Tc2_System.T_MaxString;
	returnValue			: BOOL;
END_VAR
IF previousMethodName <> methodName THEN
	returnValue := FALSE;
END_IF

IF NOT returnValue AND_THEN MemoryHelper.GetRouterStatusInfo('', _routerInfoBeforeTestMethod) THEN
	returnValue := TRUE;
END_IF

previousMethodName := methodName;
BeforeTestStart := returnValue;
END_METHOD

METHOD Test01_ProvideIncorrectParameters_ExpectNoAllocation
VAR_INPUT
END_VAR
VAR
	testMallocVar	: INT;
END_VAR
VAR_INST
	assertionsDone	: BOOL;
END_VAR
IF TcUnit.TEST_ORDERED('Test01_ProvideIncorrectParameters_ExpectNoAllocation') AND_THEN 
	BeforeTestStart('Test01_ProvideIncorrectParameters_ExpectNoAllocation') 
THEN
	IF NOT assertionsDone THEN
		// Manual allocation, element size = 0
		AssertFalse(_malloc.Allocate(0, 10), 
			'If provided size of the element is 0, Allocate should return FALSE.');	
		AssertFalse(_malloc.IsAllocated,
			'IsAllocated property should be false when failing AllocateManual');
		ValidatePropertiesAfterFailedAllocation('Allocate - element size = 0');
		
		// Manual allocation, element count = 0
		AssertFalse(_malloc.Allocate(10, 0),
			'If provided number of elements is 0, Allocat should return FALSE.');	
		AssertFalse(_malloc.IsAllocated,
			'IsAllocated property should be false when failing AllocateManual');
		ValidatePropertiesAfterFailedAllocation('Allocate - element count = 0');
		
		// Manual allocation, element size = -10
		AssertFalse(_malloc.Allocate(-10, 10), 
			'If provided size of the element is -10, AllocateManual should return FALSE.');	
		AssertFalse(_malloc.IsAllocated,
			'IsAllocated property should be false when failing AllocateManual');
		ValidatePropertiesAfterFailedAllocation('Allocate - element size = -10');
		
		// Manual allocation, element count = -10
		AssertFalse(_malloc.Allocate(10, -10),
			'If provided number of elements is -10, Allocate should return FALSE.');	
		AssertFalse(_malloc.IsAllocated,
			'IsAllocated property should be false when failing AllocateManual');
		ValidatePropertiesAfterFailedAllocation('Allocate - element size = -10');
				
		// Any allocation, element count = 0
		AssertFalse(_malloc.AllocateAny(testMallocVar, 0),
			'If provided number of elements is 0, AllocateAny should return FALSE.');	
		AssertFalse(_malloc.IsAllocated,
			'IsAllocated property should be false when failing AllocateManual');		
		ValidatePropertiesAfterFailedAllocation('AllocateAny - element count = 0');
		
		
		// Any allocation, element count = -10
		AssertFalse(_malloc.AllocateAny(testMallocVar, -10),
			'If provided number of elements is 0, AllocateAny should return FALSE.');	
		AssertFalse(_malloc.IsAllocated,
			'IsAllocated property should be false when failing AllocateManual');		
		ValidatePropertiesAfterFailedAllocation('AllocateAny - element count = -10');
		assertionsDone := TRUE;
	END_IF
		
	IF BeforeTestFinish() THEN
		TcUnit.TEST_FINISHED();
	END_IF
END_IF
END_METHOD

METHOD Test02_Allocate10Integers_ExpectNoError_ValidateProperties
VAR_INPUT
END_VAR
VAR_INST
	assertionsDone	: BOOL;
END_VAR
IF TcUnit.TEST_ORDERED('Test02_Allocate10Integers_ExpectNoError_ValidateProperties') AND_THEN 
	BeforeTestStart('Test02_Allocate10Integers_ExpectNoError_ValidateProperties') 
THEN
	IF NOT assertionsDone THEN
		AssertTrue(_malloc.Allocate(SIZEOF(INT), 10),
			'Allocation of 10 integers should return TRUE.');
			
		AssertEquals_DINT(10, _malloc.Properties.NumberOfElements,
			'NumberOfElements is incorrect.');
		AssertEquals_DINT(2, _malloc.Properties.BaseTypeSize,
			'BaseTypeSize  is incorrect.');
		AssertEquals_DINT(10 * 2, _malloc.Properties.Size,
			'Size is incorrect.');
		AssertTrue(_malloc.Properties.StartAddress <> 0,
			'StartAddress should not be 0.');
		assertionsDone := TRUE;
	END_IF
		
	IF BeforeTestFinish() THEN
		TcUnit.TEST_FINISHED();
	END_IF
END_IF
END_METHOD

METHOD Test03_Free_ExpectNoMemoryAllocated
VAR_INPUT
END_VAR
VAR_INST
	assertionsDone	: BOOL;
END_VAR
IF TcUnit.TEST_ORDERED('Test03_Free_ExpectNoMemoryAllocated') AND_THEN 
	BeforeTestStart('Test03_Free_ExpectNoMemoryAllocated') 
THEN
	IF NOT assertionsDone THEN
		_malloc.Allocate(10,10);
		AssertTrue(_malloc.Free(),
			'Freeing allocated memory should return TRUE.');
			
		AssertEquals_DINT(0, _malloc.Properties.NumberOfElements,
			'NumberOfElements should be 0 after freeing.');
		AssertEquals_DINT(0, _malloc.Properties.BaseTypeSize,
			'BaseTypeSize  should be 0 after freeing.');
		AssertEquals_DINT(0, _malloc.Properties.Size,
			'Size should be 0 after freeing.');
		AssertEquals_ULINT(0, _malloc.Properties.StartAddress,
			'StartAddress should be 0 after freeing.');
		AssertFalse(_malloc.IsAllocated,
			'IsAllocated should be FALSE when freeing.');
			
		AssertFalse(_malloc.Free(),
			'If no memory is allocated, Free() should return FALSE.');
		assertionsDone := TRUE;
	END_IF
		
	IF BeforeTestFinish() THEN
		TcUnit.TEST_FINISHED();
	END_IF
END_IF
END_METHOD

METHOD Test04_SetAndGet_ExpectGetReturnsCorrectValue
VAR_INPUT
END_VAR
VAR
	data	: INT;
	result	: INT;
END_VAR
VAR_INST
	assertionsDone	: BOOL;
END_VAR
IF TcUnit.TEST_ORDERED('Test04_SetAndGet_ExpectGetReturnsCorrectValue') AND_THEN 
	BeforeTestStart('Test04_SetAndGet_ExpectGetReturnsCorrectValue') 
THEN
	IF NOT assertionsDone THEN
		_malloc.Allocate(SIZEOF(data), 5);
		
		data := 13;
		AssertTrue(_malloc.Set(2, data), 'Setting value failed.');
			
		_malloc.Get(2, result);
		AssertEquals(data, result, 'Value fetched with Get is not correct.');
		assertionsDone := TRUE;
	END_IF
	
	IF BeforeTestFinish() THEN
		TcUnit.TEST_FINISHED();
	END_IF
END_IF
END_METHOD

METHOD Test05_SetAtIncorrectIndex_ExpectFalseReturned
VAR_INPUT
END_VAR
VAR
	value	: int;
END_VAR
VAR_INST
	assertionsDone	: BOOL;
END_VAR
IF TcUnit.TEST_ORDERED('Test05_SetAtIncorrectIndex_ExpectFalseReturned') AND_THEN 
	BeforeTestStart('Test05_SetAtIncorrectIndex_ExpectFalseReturned') 
THEN
	IF NOT assertionsDone THEN
		_malloc.Allocate(SIZEOF(value),5);
		AssertFalse(_malloc.Set(5, value), 'Setting at index outside range should return FALSE.');	
		assertionsDone := TRUE;
	END_IF
	IF BeforeTestFinish() THEN 
		TcUnit.TEST_FINISHED(); 
	END_IF
END_IF
END_METHOD

METHOD Test06_GetFromIncorrectIndex_ExpectTargetValueUnchanged_MethodReturnFalse
VAR_INPUT
END_VAR

VAR
	result	: INT;
END_VAR
VAR_INST
	assertionsDone	: BOOL;
END_VAR
IF TcUnit.TEST_ORDERED('Test06_GetFromIncorrectIndex_ExpectTargetValueUnchanged_MethodReturnFalse') AND_THEN 
	BeforeTestStart('Test06_GetFromIncorrectIndex_ExpectTargetValueUnchanged_MethodReturnFalse') 
THEN
	IF NOT assertionsDone THEN
		_malloc.AllocateAny(result, 5);
		result := 5;
		AssertFalse(_malloc.Get(5, result), 
			'When getting from index outsied of allocated memory, FALSE should be returned.');
		AssertEquals_int(5,result,
			'Getting from outside the bounds of allocated memory area, result variable should not be changed.');
		assertionsDone := TRUE;
	END_IF
	IF BeforeTestFinish() THEN
		TcUnit.TEST_FINISHED();
	END_IF
END_IF
END_METHOD

METHOD Test07_Expand_ExpectOldDataStillExists_LastDataSetIsEmpty
VAR_INPUT
END_VAR
VAR
	valueToSet	: INT;
	readValue	: INT;
	index		: INT;
END_VAR
VAR_INST
	assertionsDone	: BOOL;
END_VAR
IF TcUnit.TEST_ORDERED('Test07_Expand_ExpectOldDataStillExists_LastDataSetIsEmpty') AND_THEN 
	BeforeTestStart('Test07_Expand_ExpectOldDataStillExists_LastDataSetIsEmpty') 
THEN
	IF NOT assertionsDone THEN
		
		_malloc.Allocate(SIZEOF(INT), 5);
		
		FOR valueToSet := 0 TO 4 BY 1 DO
			_malloc.Set(valueToSet, valueToSet);
			_malloc.get(valueToSet, readValue);
			AssertEquals(
				Actual := readValue,
				Expected := valueToSet,
				Message := 'Incorrect allocation, further tests will fail!');
		END_FOR
		
		_malloc.Expand(3);
		AssertEquals_DINT(
			Actual := _malloc.Properties.NumberOfElements,
			Expected := 8,
			Message := 'Incorrect number of elements after expanding the allocated memory.');
		FOR index := 0 TO 4 BY 1 DO
			_malloc.Get(0,readValue);
			AssertEquals_INT(
				Actual := readValue,
				Expected := readValue,
				Message := Tc2_Standard.CONCAT(TO_STRING(index),'-th element is incorrect after expanding.'));
		END_FOR
		
		_malloc.Get(5, readValue);
		AssertEquals_INT(
			Actual := readValue,
			Expected := 0,
			Message := '5th (new) element is incorrect after expanding.');
			
		_malloc.Get(6, readValue);
		AssertEquals_INT(
			Actual := readValue,
			Expected := 0,
			Message := '6th (new) element is incorrect after expanding.');
			
		_malloc.Get(7, readValue);
		AssertEquals_INT(
			Actual := readValue,
			Expected := 0,
			Message := '7th (new) element is incorrect after expanding.');
		assertionsDone := TRUE;
	END_IF
		
	IF BeforeTestFinish() THEN
		TcUnit.TEST_FINISHED();
	END_IF
END_IF
END_METHOD

METHOD Test08_Remove_ExpectDataSetToCollapseBy1
VAR
	index		: INT;
	readValue	: INT;
END_VAR

VAR_INST
	assertionsDone	: BOOL;
END_VAR
IF TcUnit.TEST_ORDERED('Test08_Remove_ExpectDataSetToCollapseBy1') AND_THEN 
	BeforeTestStart('Test08_Remove_ExpectDataSetToCollapseBy1') 
THEN
	IF NOT assertionsDone THEN
		//[0,1,2,3,4,5]
		_malloc.Allocate(SIZEOF(INT), 6);
		FOR index := 0 TO 5 BY 1 DO
			_malloc.Set(index, index);
			_malloc.Get(index, readValue);
			AssertEquals(Expected := index, Actual := readValue, 
				Message := Tc2_Standard.CONCAT(TO_STRING(index), 'Allocation failed, further tests will fail.'));
		END_FOR
		
		// Expecting //[0,1,2,4,5]
		_malloc.Remove(3);
		AssertEquals_DINT(Expected := 5, Actual := _malloc.Properties.NumberOfElements,
			Message := 'Incorrect number of elements after rmoving the element at index 3.');
	
		_malloc.Get(0, readValue);
		AssertEquals_DINT(Expected := 0, Actual := readValue, 
			Message := '0th element has incorrect value after deleting element at 3rd index.');	
		
		_malloc.Get(1, readValue);
		AssertEquals_DINT(Expected := 1, Actual := readValue, 
			Message := '1st element has incorrect value after deleting element at 3rd index.');	
		
		_malloc.Get(2, readValue);
		AssertEquals_DINT(Expected := 2, Actual := readValue, 
			Message := '2d element has incorrect value after deleting element AT 3rd index.');	
			
			
		_malloc.Get(3, readValue);
		AssertEquals_DINT(Expected := 4, Actual := readValue, 
			Message := '3d element has incorrect value after deleting element AT 3rd index - did allocation not collapse correctly?');	
		
		_malloc.Get(4, readValue);
		AssertEquals_DINT(Expected := 5, Actual := readValue, 
			Message := '4th element has incorrect value after deleting element AT 3rd index - did allocation not collapse correctly?');	
		assertionsDone := TRUE;
	END_IF
	
	IF BeforeTestFinish() THEN
		TcUnit.TEST_FINISHED();
	END_IF
END_IF
END_METHOD

METHOD ValidatePropertiesAfterFailedAllocation
VAR_INPUT
	mallocMethodCalled	: Tc2_System.T_MaxString;
END_VAR
// Validate properties
AssertEquals_DINT(0, _malloc.Properties.BaseTypeSize,
	CONCAT(CONCAT('Calling method ', mallocMethodCalled), ' - BaseTypeSize should be 0 when failing allocation.'));
AssertEquals_DINT(0, _malloc.Properties.NumberOfElements,
	CONCAT(CONCAT('Calling method ', mallocMethodCalled), ' - NumberOfElements should be 0 when failing allocation.'));	
AssertEquals_DINT(0, _malloc.Properties.Size,
	CONCAT(CONCAT('Calling method ', mallocMethodCalled), ' - Size should be 0 when failing allocation.'));			
AssertEquals_ULINT(0, _malloc.Properties.StartAddress,
	CONCAT(CONCAT('Calling method ', mallocMethodCalled), ' - StartAddress should be 0 when failing allocation.'));
END_METHOD

END_FUNCTION_BLOCK

// ---- SOURCE/General/Memory/FB_Malloc.TcPOU
{attribute 'enable_dynamic_creation'}
// Function block for memory allocation. It only handles a single memory instance.
FUNCTION_BLOCK FB_Malloc
VAR
	_allocated	: POINTER TO BYTE;
	_properties	: ST_AllocatedMemoryProperties;
END_VAR

// Allocates the memory of size = elementSize * numberOfElements.
// If the memory allocation has already been done, Free() will be called first!
// Returns TRUE if allocation has been sucessfull - this can fail if incorrect parameters are provided (sie <= 0 or numberOfElements = 0)
METHOD Allocate : BOOL
VAR_INPUT
	elementSize			: DINT;	// Size of the element.
	numberOfElements	: DINT;	// Number of elements that will occupy the memory space.
END_VAR
IF elementSize <= 0 OR numberOfElements <= 0 THEN
	RETURN;
END_IF

Free();
_allocated := __NEW(BYTE, DINT_TO_UDINT((elementSize * numberOfElements)));

_properties.BaseTypeSize := elementSize;
_properties.NumberOfElements := numberOfElements;
_properties.Size := elementSize * numberOfElements;
_properties.StartAddress := _allocated;

Allocate := _allocated <> 0;
END_METHOD

// Allocates memory based on the provided parameters
// If the memory allocation has already been done, Free() will be called first!
METHOD AllocateAny : BOOL
VAR_INPUT
	dataType			: ANY;		// Provide the variable that will be used as base type here
	numberOfElements	: DINT;	// Number of elements that should be allocated.
END_VAR
AllocateAny :=  Allocate(dataType.diSize, numberOfElements);
END_METHOD

// Expands the current allocated memory
METHOD Expand : BOOL
VAR_INPUT
	elementsToAdd	: DINT; // Number of new elements to be added. Only accepting values larger than 0.
END_VAR
VAR
	oldAllocatedMemory	: POINTER TO BYTE;
	originalProperties	: ST_AllocatedMemoryProperties;
END_VAR
IF NOT IsAllocated OR elementsToAdd <= 0 THEN
	RETURN;
END_IF

// Copy current contents
originalProperties := _properties;
oldAllocatedMemory := __NEW(BYTE, (DINT_TO_UDINT(_properties.Size)));

Tc2_System.MEMCPY(
	srcAddr := _allocated, 
	destAddr := oldAllocatedMemory,
 	n := DINT_TO_UDINT(_properties.Size));

// Free the memory	
THIS^.Free();

// Create new, expanded memory
THIS^.Allocate(
	elementSize := originalProperties.BaseTypeSize ,
	numberOfElements:=  originalProperties.NumberOfElements + elementsToAdd);
	
// Copy the old values to the new allocation.	
Tc2_System.MEMCPY(
	srcAddr := oldAllocatedMemory,
	destAddr := _allocated,
	n := DINT_TO_UDINT(originalProperties.Size));
	
// Delete the temporary allocated memory
__DELETE(oldAllocatedMemory);
END_METHOD

METHOD FB_exit : BOOL
VAR_INPUT
	bInCopyCode : BOOL; // if TRUE, the exit method is called for exiting an instance that is copied afterwards (online change).
END_VAR
Free();
END_METHOD

METHOD FB_init : BOOL
VAR_INPUT
	bInitRetains : BOOL; // if TRUE, the retain variables are initialized (warm start / cold start)
	bInCopyCode : BOOL;  // if TRUE, the instance afterwards gets moved into the copy code (online change)
	baseTypeSize	: DINT;	// Base data type's that will be used
	elementCount	: DINT;	// Number of elements
END_VAR
Allocate(baseTypeSize, elementCount);
END_METHOD

// Frees the allocated memory area. 
// Returns TRUE if operation was executed (if nothing is allocated, then FALSE is returned).
METHOD Free : BOOL
VAR_INPUT
END_VAR
IF _allocated <> 0 THEN
	__DELETE(_allocated);
	_properties.BaseTypeSize := 0;
	_properties.NumberOfElements := 0;
	_properties.Size := 0;
	_properties.StartAddress := 0;
	Free := TRUE;
	RETURN;
END_IF
END_METHOD

// Gets the value at the provided 'index' copies it to the 'result' variable.
METHOD Get : BOOL
VAR_INPUT
	index	: DINT;
	result	: ANY;
END_VAR
IF NOT ValidateAction(index,result) THEN
	Get := FALSE;
	RETURN;
END_IF

Tc2_System.MEMCPY(
	destAddr := result.pValue,	
	srcAddr := _properties.StartAddress + DINT_TO_UDINT(index * _properties.BaseTypeSize),
	n := DINT_TO_UDINT(_properties.BaseTypeSize));
	
Get := TRUE;
END_METHOD

// Gets the pointer to the provided index
// This can be used to alter the contents by using POINTER TO <DATA_TYPE>. by calling it from another method
METHOD GetPtr : PVOID
VAR_INPUT
	index	: DINT;
END_VAR
IF THIS^.ValidateIndex(index) AND 
   THIS^.IsAllocated 
THEN
	GetPtr := _properties.StartAddress + DINT_TO_UDINT(index * _properties.BaseTypeSize);
END_IF
END_METHOD

{attribute 'monitoring':='call'}
// Returns TRUE if memory has been allocated.
PROPERTY PUBLIC IsAllocated : BOOL
GET
IsAllocated := _properties.StartAddress  <> 0;
END_GET
END_PROPERTY

{attribute 'monitoring':='call'}
// Gets properties of the allocated memory.
PROPERTY Properties : REFERENCE TO ST_AllocatedMemoryProperties
GET
Properties REF= _properties;
END_GET
END_PROPERTY

// Removes the element at the index.
METHOD Remove	: BOOL;
VAR_INPUT
	index	: DINT;
END_VAR

VAR
	byteCountLowerPart	: DINT;
	byteCountUpperPart	: DINT;
	upperPart			: POINTER TO BYTE;
	lowerPart			: POINTER TO BYTE;
	originalProperties	: ST_AllocatedMemoryProperties;
	newSize				: DINT;
	combinedSize		: DINT;
END_VAR
IF NOT IsAllocated OR NOT ValidateIndex(index) THEN
	RETURN;
END_IF

// If 0th element is the only element, then just free the memory space.
IF index = 0 AND _properties.NumberOfElements = 1 THEN
	Remove := TRUE;
	THIS^.Free();
	RETURN;
END_IF

originalProperties := _properties;
byteCountLowerPart := _properties.BaseTypeSize * index;
lowerPart := __NEW(BYTE, DINT_TO_UDINT(byteCountLowerPart));
Tc2_System.MEMCPY(
	srcAddr := _allocated,
	destAddr := lowerPart,
	n := DINT_TO_UDINT(byteCountLowerPart));
	
byteCountUpperPart := _properties.BaseTypeSize * (_properties.NumberOfElements - 1 - index );
IF byteCountUpperPart <> 0 THEN
	upperPart := __NEW(BYTE, DINT_TO_UDINT(byteCountUpperPart));
	Tc2_System.MEMCPY(
		srcAddr := _allocated + DINT_TO_DWORD(_properties.Size) -  DINT_TO_DWORD(byteCountUpperPart),
		destAddr := upperPart,
		n := DINT_TO_UDINT(byteCountUpperPart));	
END_IF

THIS^.Free();

// For debug purpose, new size and combined size should be the same.
newSize := originalProperties.NumberOfElements - 1;
combinedSize := (byteCountLowerPart + byteCountUpperPart) / originalProperties.BaseTypeSize;

THIS^.Allocate(originalProperties.BaseTypeSize, newSize);
Tc2_System.MEMCPY(
	srcAddr := lowerPart,
	destAddr := _allocated,
	n := DINT_TO_UDINT(byteCountLowerPart));
	
IF byteCountUpperPart <> 0 THEN
	Tc2_System.MEMCPY(
		srcAddr := upperPart,
		destAddr := _allocated + DINT_TO_UDINT(byteCountLowerPart),
		n := DINT_TO_UDINT(byteCountUpperPart));
END_IF	
	
__DELETE(lowerPart);	
IF upperPart <> 0 THEN
	__DELETE(upperPart);
END_IF

Remove := TRUE;
END_METHOD

METHOD Set : BOOL
VAR_INPUT
	index	: DINT;
	value	: ANY;
END_VAR
IF NOT ValidateAction(index,value) THEN
	Set := FALSE;
	RETURN;
END_IF

Tc2_System.MEMCPY(
	destAddr := _properties.StartAddress + DINT_TO_UDINT(index * _properties.BaseTypeSize),	
	srcAddr := value.pValue,
	n := DINT_TO_UDINT(_properties.BaseTypeSize));
	
Set := TRUE;
END_METHOD

METHOD PRIVATE ValidateAction : BOOL
VAR_INPUT
	index		: DINT;
	variable	: ANY;
END_VAR
ValidateAction := ValidateIndex(index) AND ValidateInputVar(variable) AND IsAllocated;
END_METHOD

METHOD PRIVATE ValidateIndex : BOOL
VAR_INPUT
	index	: DINT;
END_VAR
ValidateIndex := index <= (_properties.NumberOfElements - 1) AND index >= 0;
END_METHOD

METHOD PRIVATE ValidateInputVar : BOOL
VAR_INPUT
	variable	: ANY;
END_VAR
ValidateInputVar := variable.diSize = _properties.BaseTypeSize;
END_METHOD

END_FUNCTION_BLOCK

// ---- SOURCE/General/Memory/MemoryHelper.TcPOU
{attribute 'hide_all_locals'}
PROGRAM MemoryHelper

VAR
	_getRouterStatusInfo : Tc2_Utilities.FB_GetRouterStatusInfo;
END_VAR

// Gets the router info and copies it to the refRouterInfo. Returns TRUE when done.
METHOD GetRouterStatusInfo : BOOL
VAR_INPUT
	netId			: Tc2_System.T_AmsNetID;
	refRouterInfo	: REFERENCE TO Tc2_Utilities.ST_TcRouterStatusInfo;
END_VAR

VAR_INST
	
END_VAR
_getRouterStatusInfo(
	bExecute := NOT _getRouterStatusInfo.bBusy,
	sNetId := netId);
	
refRouterInfo := _getRouterStatusInfo.info;
GetRouterStatusInfo := NOT _getRouterStatusInfo.bBusy;
END_METHOD

END_PROGRAM

// ---- TESTS/Test suites/FB_StringHelper_Tests.TcPOU
FUNCTION_BLOCK INTERNAL FB_StringHelper_Tests EXTENDS FB_TestSuite
VAR_INPUT
END_VAR
VAR_OUTPUT
END_VAR
VAR
END_VAR

Test01_StartsWith();
Test02_Join();
Test03_EndsWith();
Test05_Contains();
Test06_ToLowerCase_UnlimitedSize();
Test07_ToUpperCase_UnlimitedSize();

METHOD Test01_StartsWith
VAR_INPUT
END_VAR
TcUnit.TEST('Test01_StartsWith');

AssertFalse(StringHelper.StartsWith('I start with an "I"...','B'), 
	'The provided string does not start with B. Method should return FALSE.');
	
AssertTrue(StringHelper.StartsWith('I start with an "I"...','I'), 
	'The provided string start with I. Method should return TRUE..');

TcUnit.TEST_FINISHED();
END_METHOD

METHOD Test02_Join
VAR_INPUT
END_VAR

VAR
	sourceString	: Tc2_System.T_MaxString := 'My cats name is ';
END_VAR
TcUnit.TEST('Test02_Join');

StringHelper.Join(sourceString, 'Jerry');
AssertEquals_STRING('My cats name is Jerry', sourceString,
	'Joining 2 strings failed.');

TcUnit.TEST_FINISHED();
END_METHOD

METHOD Test03_EndsWith
VAR_INPUT
END_VAR

VAR
	testString	: STRING := 'I end with an A';
END_VAR
TcUnit.TEST('Test03_EndsWith');

AssertFalse(StringHelper.EndsWith(testString, 'B'),
	'Provided string does not end with "B"- returned value should be FALSE.');
AssertTrue(StringHelper.EndsWith(testString, 'A'),
	'Provided string ends with "A"- returned value should be TRUE.');
	
TcUnit.TEST_FINISHED();
END_METHOD

METHOD Test05_Contains
VAR_INPUT
END_VAR
VAR
	mainStringAsTmaxString		: Tc2_System.T_MaxString := 'asdfasdfadfasdfadfigsjcan you find mgndfkghdfghgdg!can you find me?';
	substringToFind_TmaxString	: STRING := 'can you find me';
	mainStringAsString300		: STRING(300) := 
		'abcdefghijklmnopqrstuvwxyzABCDEFGHIJKLMNOPQRSTUVWXYZ0123456789abcdefghijklmThis is the test sentence.nopqrstuvwxyzABCDEFGHIJKLMNOPQRSTUVWXYZ0123456789abcdefghijklmnopqrstuvwxyzABCDEFGHIJKLMNOPQRSTUVWXYZ0123456789abcdefghijklmnopqrstuvwxyz';
	substringToFind_String300	: STRING := 'This is the test sentence';	
	mainStringTmp				: STRING(300);
	position 					: DINT;
	test	: int;
END_VAR
TcUnit.TEST('Test05_Contains');

// T_MaxString tests

// doesen't contain
AssertFalse(StringHelper.FindStringWithin(mainStringAsTmaxString, 'test123', position => position),
	'String does not contain the provided substring.');
AssertEquals_DINT(0, position,
	'When string is not found, position should be 0');

// Upper case - fail
AssertFalse(StringHelper.FindStringWithin(mainStringAsTmaxString, StringHelper.ToUpperCase(substringToFind_TmaxString), position => position),
	'String should not be found, provided string is in upper case.');
AssertEquals_DINT(0, position,
	'When string is not found (upper case) , position should be 0');

// Contains	
AssertTrue(StringHelper.FindStringWithin(mainStringAsTmaxString, substringToFind_TmaxString, position => position),
	'String contains the provided substring, expected returned value should be TRUE.');
AssertEquals_DINT(52, position,
	'Incorrect position of the found substring.');
	

// Strings larger than T_MaxString tests
// Does not contain
AssertFalse(StringHelper.FindStringWithin(mainStringAsString300, 'test1234', position => position),
	'String300 - provided substring does not exist in the main string, expected FALSE.');
AssertEquals_DINT(0, position,
	'String300 - when substring is not found, expected position is 0.');
	
// Upper case - fail	
mainStringTmp := mainStringAsString300;
StringHelper.ToUpperCase_UnlimitedSize(mainStringTmp);
AssertFalse(StringHelper.FindStringWithin(mainStringAsTmaxString, mainStringTmp, position => position),
	'String300 upper case - String should not be found, provided string is in upper case.');
AssertEquals_DINT(0, position,
	'String300 upper case - When string is not found (upper case) , position should be 0');
	
// Lower case - fail
mainStringTmp := mainStringAsString300;
StringHelper.ToLowerCase_UnlimitedSize(mainStringTmp);
AssertFalse(StringHelper.FindStringWithin(mainStringAsTmaxString, mainStringTmp, position => position),
	'String300 lower case - String should not be found, provided string is in lower case.');
AssertEquals_DINT(0, position,
	'String300 lower case - When string is not found (lower case), position should be 0');
test := Tc2_Standard.FIND(mainStringAsString300, substringToFind_String300);
// Contains	
AssertTrue(StringHelper.FindStringWithin(mainStringAsString300, substringToFind_String300, position => position),
	'String contains the provided substring, expected returned value should be TRUE.');
AssertEquals_DINT(76, position,
	'Incorrect position of the found substring.');	
	
TcUnit.TEST_FINISHED();
END_METHOD

METHOD Test06_ToLowerCase_UnlimitedSize
VAR_INPUT
END_VAR
VAR_INST
	expectedResult	: STRING(300) := 'abcdefghijklmnopqrstuvwxyzabcdefghijklmnopqrstuvwxyz0123456789abcdefghijklmthis is the test sentence.nopqrstuvwxyzabcdefghijklmnopqrstuvwxyz0123456789abcdefghijklmnopqrstuvwxyzabcdefghijklmnopqrstuvwxyz0123456789abcdefghijklmnopqrstuvwxyz';
	providedString	: STRING(300) := 'ABCDEFGHIJKLMNOPQRSTUVWXYZABCDEFGHIJKLMNOPQRSTUVWXYZ0123456789ABCDEFGHIJKLMTHIS IS THE TEST SENTENCE.NOPQRSTUVWXYZABCDEFGHIJKLMNOPQRSTUVWXYZ0123456789ABCDEFGHIJKLMNOPQRSTUVWXYZABCDEFGHIJKLMNOPQRSTUVWXYZ0123456789ABCDEFGHIJKLMNOPQRSTUVWXYZ';
END_VAR
TcUnit.TEST('Test06_ToLowerCase_UnlimitedSize');

StringHelper.ToLowerCase_UnlimitedSize(providedString);
AssertEquals(expectedResult, providedString,
	'Incorrect conversion to lower case of string(300)');
	
TcUnit.TEST_FINISHED();
END_METHOD

METHOD Test07_ToUpperCase_UnlimitedSize
VAR_INPUT
END_VAR
VAR_INST
	providedString	: STRING(300) := 'abcdefghijklmnopqrstuvwxyzABCDEFGHIJKLMNOPQRSTUVWXYZ0123456789abcdefghijklmThis is the test sentence.nopqrstuvwxyzABCDEFGHIJKLMNOPQRSTUVWXYZ0123456789abcdefghijklmnopqrstuvwxyzABCDEFGHIJKLMNOPQRSTUVWXYZ0123456789abcdefghijklmnopqrstuvwxyz';
	expectedResult	: STRING(300) := 'ABCDEFGHIJKLMNOPQRSTUVWXYZABCDEFGHIJKLMNOPQRSTUVWXYZ0123456789ABCDEFGHIJKLMTHIS IS THE TEST SENTENCE.NOPQRSTUVWXYZABCDEFGHIJKLMNOPQRSTUVWXYZ0123456789ABCDEFGHIJKLMNOPQRSTUVWXYZABCDEFGHIJKLMNOPQRSTUVWXYZ0123456789ABCDEFGHIJKLMNOPQRSTUVWXYZ';
END_VAR
TcUnit.TEST('Test07_ToUpperCase_UnlimitedSize');

StringHelper.ToUpperCase_UnlimitedSize(providedString);
AssertEquals(expectedResult, providedString,
	'Incorrect conversion to upper case of string(300)');
	
TcUnit.TEST_FINISHED();
END_METHOD

END_FUNCTION_BLOCK

// ---- SOURCE/String/StringHelper.TcPOU
PROGRAM StringHelper
VAR
END_VAR

METHOD EndsWith : BOOL
VAR_INPUT
	str		: Tc2_System.T_MaxString;
	char	: T_Char;	
END_VAR
EndsWith := Tc2_Standard.RIGHT(str, 1) = char;
END_METHOD

// Checks if the sourceString contains the stringToFind string. 
// Size of the source string is only limited to TwinCAT limitaitons, which in theory is not limited.
// Returns TRUE if found, else FALSE. Position of the found strimg is provided in the "position" output variable.
METHOD FindStringWithin : BOOL
VAR_INPUT
	sourceString	: ANY;	// String to look at
	stringToFind	: Tc2_System.T_MaxString; // String that should be containted in the sourceString
END_VAR
VAR_OUTPUT
	position	: DINT;	// Position of the found string
END_VAR

VAR
	tmpStr						: POINTER TO Tc2_System.T_MaxString;
	charIndex					: DINT;
	currentMatchingCharIndex	: DINT;
	tmpByte						: POINTER TO BYTE;
	firstCharPosition 			: dint;
END_VAR
IF NOT F_DoesVarTypeEqual(sourceString, IBaseLibrary.TYPE_STRING) THEN
	RETURN;
END_IF

IF sourceString.diSize <= SIZEOF(Tc2_System.T_MaxString) THEN
	tmpStr := __NEW(BYTE, SIZEOF(Tc2_System.T_MaxString));
	Tc2_System.MEMCPY(
		destAddr := tmpStr,
		srcAddr := sourceString.pValue,
		n := DINT_TO_UDINT(sourceString.diSize));
	//tmpStr := sourceString.pValue;
	position :=  Tc2_Standard.FIND(tmpStr^, stringToFind);
	FindStringWithin := position <> 0;
	__DELETE(tmpStr);
	RETURN;
END_IF

FOR charIndex := 0 TO sourceString.diSize BY 1 DO
	
	// Byte wise comparison, if matching byte, start filling the compared string
	tmpByte := sourceString.pValue + charIndex * SIZEOF(BYTE);
	// For debug purpose
	tmpStr := tmpByte;
	IF tmpbyte^ = stringToFind[currentMatchingCharIndex] THEN
		IF firstCharPosition = 0 THEN
			firstCharPosition := charIndex + 1;
		END_IF
		currentMatchingCharIndex := currentMatchingCharIndex + 1;
	ELSE
		currentMatchingCharIndex := 0;
		firstCharPosition := 0;
	END_IF
	
	// When index = str lenght - 1, we have found the entire string, exit the loop.
	IF currentMatchingCharIndex = (Tc2_Standard.LEN(stringToFind)) THEN
		position := firstCharPosition;
		FindStringWithin := TRUE;
		EXIT;
	END_IF
END_FOR
END_METHOD

// Joins the provided string with the string to add.
// The refStr is altered in the process, this no additional assignments are required as oposed to CONCAT which returns the resulting string.
METHOD Join
VAR_INPUT
	refStr		: REFERENCE TO Tc2_System.T_MaxString;
	strToJoin	: Tc2_System.T_MaxString;
END_VAR
refStr := Tc2_Standard.CONCAT(refStr, strToJoin);
END_METHOD

// Checks if STRING `str` starts with the `char`
// Returs TRUE if first character in the provided string is `char` provided
METHOD StartsWith : BOOL
VAR_INPUT
	str		: Tc2_System.T_MaxString;	// String to be checked
	char	: T_Char;	// Character that the string will be checked, if it starts with it.
END_VAR
StartsWith := Tc2_System.F_ToCHR(str[0]) = char;
END_METHOD

// Converts the provided string to all lower case and returns the converted value.
METHOD ToLowerCase : T_MaxString
VAR_INPUT
	str	: Tc2_System.T_MaxString;	// Source string
END_VAR
ToLowerCase := Tc2_Utilities.F_ToLCase(in := str);
END_METHOD

// Converts the input string to all lower case. Size of the string is irrelevant
METHOD ToLowerCase_UnlimitedSize
VAR_INPUT
	str	: ANY;
END_VAR

VAR
	charIndex	: DINT;
	ptrChar		: POINTER TO T_Char;
	char		: T_Char;
	malloc		: FB_Malloc(0,0);
	ptrByte		: POINTER TO BYTE;
END_VAR
IF NOT F_DoesVarTypeEqual(str, IBaseLibrary.TYPE_STRING) THEN
	RETURN;
END_IF

malloc.Allocate(1, str.diSize - 1);		
FOR charIndex := 0 TO str.diSize - 1 BY 1 DO
	ptrChar := str.pValue + DINT_TO_DWORD(charIndex);
	char := ToLowerCase(ptrChar^);
	ptrByte := ADR(char);
	malloc.Set(charIndex, ptrByte^);
END_FOR

Tc2_System.MEMCPY(
	destAddr := str.pValue, 
	srcAddr := malloc.Properties.StartAddress, 
	n := DINT_TO_UDINT(str.diSize - 1));
	
malloc.Free();
END_METHOD

// Converts the provided string to all upper case and returns the converted value.
METHOD ToUpperCase : Tc2_System.T_MaxString
VAR_INPUT
	str	: Tc2_System.T_MaxString;	// Source string
END_VAR
ToUpperCase := Tc2_Utilities.F_ToUCase(in := str);
END_METHOD

METHOD ToUpperCase_UnlimitedSize
VAR_INPUT
	str	: ANY;
END_VAR	

VAR
	charIndex	: DINT;
	ptrChar		: POINTER TO T_Char;
	char		: T_Char;
	malloc		: FB_Malloc(0,0);
	ptrByte		: POINTER TO BYTE;
END_VAR
IF NOT F_DoesVarTypeEqual(str, IBaseLibrary.TYPE_STRING) THEN
	RETURN;
END_IF

malloc.Allocate(1, str.diSize - 1);		
FOR charIndex := 0 TO str.diSize - 1 BY 1 DO
	ptrChar := str.pValue + DINT_TO_DWORD(charIndex);
	char := ToUpperCase(ptrChar^);
	ptrByte := ADR(char);
	malloc.Set(charIndex, ptrByte^);
END_FOR

Tc2_System.MEMCPY(
	destAddr := str.pValue, 
	srcAddr := malloc.Properties.StartAddress, 
	n := DINT_TO_UDINT(str.diSize - 1));
	
malloc.Free();
END_METHOD

// Removes leading spaces from the character string and returns the reduced character string
METHOD PUBLIC TrimLeftSide : Tc2_System.T_MaxString
VAR_INPUT
	str	: Tc2_System.T_MaxString; // String to be trimmed
END_VAR
TrimLeftSide := Tc2_Utilities.F_LTrim(in := str);
END_METHOD

// Truncates all trailing spaces from the specified value and returns the result.
METHOD PUBLIC TrimRightSide : Tc2_System.T_MaxString
VAR_INPUT
	str	: Tc2_System.T_MaxString;	// String to be trimmed
END_VAR
TrimRightSide := Tc2_Utilities.F_RTrim(in := str);
END_METHOD

END_PROGRAM

// ---- TESTS/Test suites/Time/FB_LocalSystemTime_Tests.TcPOU
FUNCTION_BLOCK INTERNAL FB_LocalSystemTime_Tests EXTENDS TcUnit.FB_TestSuite
VAR_INPUT
END_VAR
VAR_OUTPUT
END_VAR
VAR
	_localSystemTimeProvider	: FB_LocalSystemTimeProvider;
END_VAR

_localSystemTimeProvider();
Test01_CheckSystemTime_ExpectValue();
Test02_SetSystemTime_ExpectNoErrorAndCorrectTimeRead();

METHOD Test01_CheckSystemTime_ExpectValue
VAR_INPUT
END_VAR

VAR
	emptyTimeStruct	: Tc2_Utilities.TIMESTRUCT;
END_VAR

IF TcUnit.TEST_ORDERED('Test01_CheckSystemTime_ExpectValue') THEN
	IF _localSystemTimeProvider.CurrentTime.IsValid THEN
		AssertTrue(
			Tc2_System.MEMCMP(ADR(emptyTimeStruct),
				ADR(_localSystemTimeProvider.CurrentTime.Value), 
				SIZEOF(Tc2_Utilities.TIMESTRUCT)) <> E_MemCmpResults.IDENTICAL,
			'System time returned an empty property value!');
		TcUnit.TEST_FINISHED();		
	END_IF
END_IF
END_METHOD

METHOD PRIVATE Test02_SetSystemTime_ExpectNoErrorAndCorrectTimeRead
VAR_INPUT
END_VAR
VAR CONSTANT
	timeToSet	: Tc2_Utilities.TIMESTRUCT := (
		wYear := 2026, 
		wMonth := 2, 
		wDay := 3, 
		wHour := 4,
		wMinute := 5,
		wSecond := 5,
		wMilliseconds := 7);
END_VAR
VAR
	error	: BOOL;
	errorId	: TcError.AdsErrorCodes;
END_VAR
VAR_INST
	testAssertionsDone_WaitForSystemTimeToBeSetBackToOriginalValue	: BOOL;
	originalTime	: Tc2_Utilities.TIMESTRUCT;
	timeSettingDone		: BOOL;
	waitForSynchronisationOfLocalSystemTime		: Tc2_Standard.TON := (PT := T#1200MS);
END_VAR
IF TcUnit.TEST_ORDERED('Test02_SetSystemTime_ExpectNoErrorAndCorrectTimeRead') THEN
	IF _localSystemTimeProvider.CurrentTime.IsValid THEN
		// Save original time to reset due to TwinCAT licensing system
		IF originalTime.wYear = 0 THEN
			originalTime := _localSystemTimeProvider.CurrentTime.Value;			
		END_IF
		
		// Set time only once
		IF NOT timeSettingDone AND_THEN _localSystemTimeProvider.SetSystemTime(timeToSet, error => error, errorId => errorId ) THEN
			waitForSynchronisationOfLocalSystemTime.IN := TRUE;
			AssertFalse(error, 
				'Error occured attempting to set system time');
			AssertTrue(errorId = TcError.AdsErrorCodes.ERR_NOERROR, 
				CONCAT('Error has occured - ', TO_STRING(errorId)));
			timeSettingDone := TRUE;				
		END_IF
		
		waitForSynchronisationOfLocalSystemTime(IN := timeSettingDone);
		// Since dwCycle minimum setting is 1 second (DWORD, seconds), we need to wait before we have a valid time value
		
		IF waitForSynchronisationOfLocalSystemTime.Q AND NOT 
			testAssertionsDone_WaitForSystemTimeToBeSetBackToOriginalValue 
		THEN
			AssertEquals_WORD(_localSystemTimeProvider.CurrentTime.Value.wYear, 2026, 'Year was not set correctly!');
			AssertEquals_WORD(_localSystemTimeProvider.CurrentTime.Value.wMonth, 2, 'Month was not set correctly!');
			AssertEquals_WORD(_localSystemTimeProvider.CurrentTime.Value.wDay, 3, 'Day was not set correctly!');
			AssertEquals_WORD(_localSystemTimeProvider.CurrentTime.Value.wHour, 4, 'Hour was not set correctly!');
			AssertEquals_WORD(_localSystemTimeProvider.CurrentTime.Value.wMinute, 5, 'Minute was not set correctly!');
			// Since synchronisation is done with 1 second (minimum), check the value range for second and millisecond
			AssertTrue(_localSystemTimeProvider.CurrentTime.Value.wSecond >= 6, 'Second was not set correctly!');
			AssertTrue(_localSystemTimeProvider.CurrentTime.Value.wMilliseconds >= 7, 'Millisecond was not set correctly!');
			testAssertionsDone_WaitForSystemTimeToBeSetBackToOriginalValue := TRUE;
		END_IF
		
		// Set time back othewise TwinCAT stops working due to invalid license :)
		IF testAssertionsDone_WaitForSystemTimeToBeSetBackToOriginalValue THEN
			IF _localSystemTimeProvider.SetSystemTime(originalTime) THEN
				TcUnit.TEST_FINISHED();	
			END_IF
		END_IF
	END_IF
END_IF
END_METHOD

END_FUNCTION_BLOCK

// ---- SOURCE/Time/FB_LocalSystemTimeProvider.TcPOU
FUNCTION_BLOCK FB_LocalSystemTimeProvider IMPLEMENTS I_LocalSystemTimeProvider
VAR
	_localSystemTime			: Tc2_Utilities.FB_LocalSystemTime;
	_currentSystemTimeInfo		: ST_CurrentSystemTimeInfo;
	_dateTimeToStringCovnerter	: FB_DateTimeToStringConverter;
	_iDateTimeToStringConverter	: I_DateTimeToStringConverter := _dateTimeToStringCovnerter;
END_VAR

_localSystemTime(
	sNetID:= '', 
	bEnable:= TRUE, 
	dwCycle:= 1, 
	systemTime=> _currentSystemTimeInfo.Value);
	
_currentSystemTimeInfo.IsValid := _currentSystemTimeInfo.Value.wYear > 1970;
	
_dateTimeToStringCovnerter(
	localSystemTime := _localSystemTime);

METHOD PUBLIC ConvertToString : I_DateTimeToStringConverter
VAR_INPUT
END_VAR
ConvertToString := _iDateTimeToStringConverter;
END_METHOD

{attribute 'monitoring':='call'}
// Gets current system timo info as a <ST_CurrentSystemTimeInfo>
PROPERTY CurrentTime : REFERENCE TO ST_CurrentSystemTimeInfo
GET
CurrentTime REF= _currentSystemTimeInfo;
END_GET
END_PROPERTY

// Sets the system time. Returns TRUE when done.
METHOD SetSystemTime : BOOL
VAR_INPUT
	timeToSet	: Tc2_Utilities.TIMESTRUCT;
END_VAR

VAR_OUTPUT
	error	: BOOL;	// Will be TRUE if an error occurs
	errorId	: TcError.AdsErrorCodes;	// Error code is reported here
END_VAR

VAR_INST
	setLocalTime	: Tc2_Utilities.NT_SetLocalTime :=(
		NETID := '',
		TMOUT := Tc2_System.DEFAULT_ADS_TIMEOUT);
END_VAR
setLocalTime(
	START := NOT setLocalTime.BUSY, 
	TIMESTR := timeToSet,
	ERR => error);
	
errorId := TcError.ToAdsErrorCode(TcError.ToAdsErrorCode(setLocalTime.ERRID));
SetSystemTime := NOT setLocalTime.BUSY;
END_METHOD

END_FUNCTION_BLOCK

// ---- TESTS/Test suites/FB_CoeReadWrite_Tests.TcPOU
FUNCTION_BLOCK INTERNAL FB_CoeReadWrite_Tests EXTENDS FB_TestSuite
VAR_INPUT
END_VAR
VAR_OUTPUT
END_VAR
VAR
	_coeReadWrite			: FB_CoeReadWrite();
	_coeReadWriteError		: BOOL;
	_coeReadWriteErorId		: TcError.AdsErrorCodes;
	_coeDeviceAmsAddress	: Global.AMSADDR;
	_coeEntry				: ST_CoeEntry_DINT();
END_VAR

Test00_ReadAny_ExpectError();
Test01_WriteAny_ExpectError();

METHOD PRIVATE Test00_ReadAny_ExpectError
IF TcUnit.TEST_ORDERED(__POUNAME()) THEN
	IF _coeReadWrite.ReadAny(ADR(_coeEntry), _coeEntry.Value, _coeDeviceAmsAddress, error => _coeReadWriteError, errorId => _coeReadWriteErorId) THEN
		AssertTrue(
			Condition := _coeReadWriteError,
			Message := 'Reading an invalid slave COE should return an error!');
			TcUnit.TEST_FINISHED();
	END_IF
END_IF
END_METHOD

METHOD PRIVATE Test01_WriteAny_ExpectError
VAR_INPUT
END_VAR
VAR
	valueToWrite	: DINT;
END_VAR
IF TcUnit.TEST_ORDERED(__POUNAME()) THEN
	IF _coeReadWrite.WriteAny(ADR(_coeEntry), valueToWrite, _coeDeviceAmsAddress, error => _coeReadWriteError, errorId => _coeReadWriteErorId) THEN
		AssertTrue(
			Condition := _coeReadWriteError,
			Message := 'Writing to invalid slave COE should return an error');
		TcUnit.TEST_FINISHED();
	END_IF
END_IF
END_METHOD

END_FUNCTION_BLOCK

// ---- SOURCE/Beckhoff/EtherCAT/CoE/FB_CoeReadWrite.TcPOU
FUNCTION_BLOCK FB_CoeReadWrite
VAR
END_VAR

// Reads the CoE parameter at Index:Subindex and writes the value to Value. Returns TRUE when done.
METHOD PUBLIC ReadAny : BOOL
VAR_INPUT
	CoeEntry	: POINTER TO ST_CoeEntry;	// Pointer to CoE entry, index and subindex
	Value		: ANY;						// Value to where the read result is stored (you can use extended ST_CoeEntry_<DataType> from the library
	SlaveAddr	: Global.AMSADDR;			// Slave AMS address of the device
END_VAR

VAR_OUTPUT
	error	: BOOL;						// Will be TRUE if the reading failed
	errorId	: TcError.AdsErrorCodes;	// Error ID when an error has occured.
END_VAR

VAR_INST
	fbCoeRead		: Tc2_EtherCAT.FB_EcCoESdoRead;
	FtrigReadDone	: Tc2_Standard.F_TRIG;
END_VAR
fbCoeRead(
	sNetId:= AdsHelper.NetIdToString(SlaveAddr.netId), 
	nSlaveAddr:= SlaveAddr.port, 
	nSubIndex:= CoeEntry^.Subindex, 
	nIndex:= CoeEntry^.Index, 
	pDstBuf:= Value.pValue, 
	cbBufLen:= DINT_TO_UDINT(Value.diSize), 
	bExecute:= NOT fbCoeRead.bBusy, 
	tTimeout:= T#5S, 
	bError=> error);
	
errorId := TcError.ToAdsErrorCode(fbCoeRead.nErrId);
FtrigReadDone(CLK := fbCoeRead.bBusy);
ReadAny := FtrigReadDone.Q;
END_METHOD

// Writes the CoE parameter at Index:Subindex and returns TRUE when done.
METHOD WriteAny : BOOL
VAR_INPUT
	CoeEntry	: POINTER TO ST_CoeEntry;	// Pointer to CoE entry, index and subindex
	Value		: ANY;						// Value that should be written to the CoE entry
	SlaveAddr	: Global.AMSADDR;					// Slave AMS address of the device
END_VAR

VAR_OUTPUT
	error	: BOOL;						// Will be TRUE if the writing failed
	errorId	: TcError.AdsErrorCodes;	// Error ID when an error has occured.
END_VAR

VAR_INST
	fbCoeWrite		: Tc2_EtherCAT.FB_EcCoESdoWrite;
	FtrigWriteDone	: Tc2_Standard.F_TRIG;
END_VAR
fbCoeWrite(
	sNetId:= AdsHelper.NetIdToString(SlaveAddr.netId), 
	nSlaveAddr:= SlaveAddr.port, 
	nSubIndex:= CoeEntry^.Subindex,
	nIndex:= CoeEntry^.Index, 
	pSrcBuf:= Value.pValue, 
	cbBufLen:= DINT_TO_UDINT(Value.diSize), 
	bExecute:= NOT fbCoeWrite.bBusy, 
	tTimeout:= T#3S,
	bError => error,);
	
errorId := TcError.ToAdsErrorCode(errorCode := fbCoeWrite.nErrId);
FtrigWriteDone(CLK := fbCoeWrite.bBusy, Q => WriteAny);
END_METHOD

END_FUNCTION_BLOCK

// ---- SOURCE/Beckhoff/Ads/FB_HasAmsAddressFromProcessImage.TcPOU
// Inherit from this FB to get Tc2_System.ST_AmsAddr in the process image (to link to EtherCAT devices etc...)
FUNCTION_BLOCK ABSTRACT FB_HasAmsAddressFromProcessImage
VAR_INPUT
END_VAR
VAR_OUTPUT
END_VAR
VAR
	Ams AT%I* 	: Tc2_System.ST_AmsAddr;
	_ams 		: Tc2_System.ST_AmsAddr;
END_VAR

(* Gets or sets the Ams address structure*)
PROPERTY AmsAddress : REFERENCE TO Tc2_System.ST_AmsAddr
GET
_ams := Ams;
AmsAddress REF= _ams;
END_GET
END_PROPERTY

END_FUNCTION_BLOCK

// ---- SOURCE/Beckhoff/EtherCAT/Diagnosis/FB_EthercatDiagnosis.TcPOU
// Function block for EtherCAT diagnosis, looking at the live slave status and reporting back any missing slaves
FUNCTION_BLOCK FB_EthercatDiagnosis IMPLEMENTS I_EthercatDiagnosis
VAR
	_ignoredSlaves	: ARRAY[0..255] OF Tc2_System.T_MaxString;
	_missingSlaves	: ARRAY[0..255] OF ST_EthercatSlaveInfo;
	_status			: E_EthercatDiagnosisStatus;
	_diagState		: E_EthercatDiagnosisState;
	_error			: BOOL;
END_VAR

(* Returns TRUE if an error occurred while performing the scan*)
PROPERTY Error : BOOL
GET
Error := _error;
END_GET
END_PROPERTY

(* Gets an array of slaves that have been added to ignore list*)
PROPERTY IgnoredSlaves : REFERENCE TO ARRAY [0..255] OF Tc2_System.T_MaxString
GET
IgnoredSlaves REF= _ignoredSlaves;
END_GET
END_PROPERTY

(* Adds the provided slave to a collection of slaves that will not trigger an error
 Example is slaves that are used on hot connect groups, and when connected should not cause an error. *)
METHOD IgnoreSlave
VAR_INPUT
	(* Slave to be ignored if not found or an error is reported back*)
	name	: Tc2_System.T_MaxString;
END_VAR
IF name <> '' THEN
	ArrayHelper.InsertAtStart(arr := _ignoredSlaves, item := name);
END_IF
END_METHOD

(* Returns an array of misisng slave names*)
PROPERTY MissingSlaves : REFERENCE TO ARRAY [0..255] OF ST_EthercatSlaveInfo
GET
MissingSlaves REF= _missingSlaves;
END_GET
END_PROPERTY

{warning 'add method implementation '}
(* Reset the internal state machine of diagnosis and clearing any errors, if active.*)
METHOD Reset
END_METHOD

{warning 'add method implementation '}
(* Performs a scan on the EtherCAT master, returns TRUE when done.*)
METHOD Scan : BOOL
VAR_INPUT
	EcMasterNetId	: AMSNETID;
END_VAR
END_METHOD

(* Gets the status based on last executed scan.*)
PROPERTY Status : E_EthercatDiagnosisStatus
GET
Status := _status;
END_GET
END_PROPERTY

END_FUNCTION_BLOCK

// ---- SOURCE/Beckhoff/EtherCAT/FB_ReadBoxName.TcPOU
// Reads box name and return string
FUNCTION_BLOCK FB_ReadBoxName
VAR_INPUT
	PlcRuntimeNetId		: Tc2_System.T_AmsNetID; // NetId of the PLC where the devuce is located
	AmsNetId			: AMSADDR; // NetId of the box
END_VAR
VAR_OUTPUT
		error 	:  BOOL;	// If an error occurs while executing, method will provide the error flag here. This is a pointer to YOUR boolean error variable.
		done		: BOOL;
		name		: Tc2_System.T_MaxString;
END_VAR

VAR
	fbReadDeviceName	: Tc2_IoFunctions.IOF_GetBoxNameByAddr;
END_VAR

fbReadDeviceName(
	NETID := PlcRuntimeNetId,
	DEVICEID := AdsHelper.GetEthercatMasterIdFromNetIdString(AdsHelper.NetIdToString(AmsNetId.netId)),
	BOXADDR := AmsNetId.port,
	START := NOT fbReadDeviceName.BUSY);
	
error := fbReadDeviceName.ERR;
name := fbReadDeviceName.BOXNAME;

END_FUNCTION_BLOCK

// ---- SOURCE/General/FB_BooleanObserver.TcPOU
// Boolean condition observer. Body requires calling every cycle in order to execute the triggers!
// Checkes the "bCondition" and returns a 1 cycle pulse output on bRisingEdge when value changes form 0 to 1
// Checkes the "bCondition" and returns a 1 cycle pulse output on bFallingEdge when value changes form 1 to 0

FUNCTION_BLOCK FB_BooleanObserver
VAR_INPUT
	bCondition	: BOOL;
END_VAR
VAR_OUTPUT
	bRisingEdge		: BOOL;
	bFallingEdge	: BOOL;
END_VAR
VAR
	_rtrig	: Tc2_Standard.R_TRIG;
	_ftrig	: Tc2_Standard.F_TRIG;
END_VAR

_rtrig(CLK := bCondition, Q => bRisingEdge);
_ftrig(CLK := bCondition, Q => bFallingEdge);

END_FUNCTION_BLOCK

// ---- SOURCE/General/FB_Watchdog.TcPOU
// A watchdog function block. Observer "variable" input - if the value does not change within the "timeout" parameter, status will return "FALSE"
FUNCTION_BLOCK FB_Watchdog
VAR_INPUT
	variable	: BOOL;	// Variable to observe
	timeout		: TIME;	// Time within the variable needs to change it's state before status is reported as FALSE
END_VAR

VAR_OUTPUT
	status	: BOOL;	// TRUE = OK, FALSE = timeout
END_VAR

VAR
	Ton_TrueTimer	: Tc2_Standard.TON;
	Ton_Falsetimer	: Tc2_Standard.TON;
END_VAR

Ton_TrueTimer(IN := variable, PT := timeout);
Ton_Falsetimer(IN := NOT variable, PT := timeout);


status := Ton_TrueTimer.Q = FALSE AND  Ton_Falsetimer.Q = FALSE;

END_FUNCTION_BLOCK

// ---- SOURCE/General/Variable information/F_GetVarInfo.TcPOU
// Returns information about the variable as ST_VarInfo.
FUNCTION F_GetVarInfo : ST_VarInfo
VAR_INPUT
	variable	: ANY;	// Variable to get the inforation from
END_VAR
VAR
END_VAR

F_GetVarInfo.Address := variable.pValue;
F_GetVarInfo.DataType := variable.TypeClass;
F_GetVarInfo.Size := DINT_TO_UDINT(variable.diSize);

END_FUNCTION

// ---- TESTS/Test suites/FB_EthercatDiagnosis_Tests.TcPOU
FUNCTION_BLOCK internal FB_EthercatDiagnosis_Tests EXTENDS FB_TestSuite
VAR_INPUT
END_VAR
VAR_OUTPUT
END_VAR
VAR
END_VAR

Test01_IgnoreSlave_ExpectSlaveInProperty();

METHOD Test01_IgnoreSlave_ExpectSlaveInProperty
VAR_INPUT
END_VAR
VAR_INST
	diag			: FB_EthercatDiagnosis;
	ignoredSlave	: Tc2_System.T_MaxString := 'I feel ignored...';
END_VAR
TcUnit.TEST('Test01_IgnoreSlave_ExpectSlaveInProperty');

diag.IgnoreSlave(ignoredSlave);
AssertTrue(
	Condition := ArrayHelper.DoesArrayContainItem(diag.IgnoredSlaves ,ignoredSlave),
	Message := 'After adding slave to ignore list, it did not appear in the .IgnoredSlaves property.');
	
TcUnit.TEST_FINISHED();
END_METHOD

END_FUNCTION_BLOCK
